(* IEC 61131-3 sources: volt/packages/volt-lsp-iec/test-corpus/lenze-mid/Device/Plc Logic/Application/Library Manager/(unresolved)/cmpopcuastack interfaces (part 4) *)

(* ---- OPCUA_BROWSENAMES.gvl ---- *)
VAR_GLOBAL
	OPCUA_BROWSENAME_3DCARTESIANCOORDINATES : STRING := '3DCartesianCoordinates';
	OPCUA_BROWSENAME_3DCARTESIANCOORDINATESTYPE : STRING := '3DCartesianCoordinatesType';
	OPCUA_BROWSENAME_3DFRAME : STRING := '3DFrame';
	OPCUA_BROWSENAME_3DFRAMETYPE : STRING := '3DFrameType';
	OPCUA_BROWSENAME_3DORIENTATION : STRING := '3DOrientation';
	OPCUA_BROWSENAME_3DORIENTATIONTYPE : STRING := '3DOrientationType';
	OPCUA_BROWSENAME_3DVECTOR : STRING := '3DVector';
	OPCUA_BROWSENAME_3DVECTORTYPE : STRING := '3DVectorType';
	OPCUA_BROWSENAME_A : STRING := 'A';
	OPCUA_BROWSENAME_ACCESSHISTORYDATACAPABILITY : STRING := 'AccessHistoryDataCapability';
	OPCUA_BROWSENAME_ACCESSHISTORYEVENTSCAPABILITY : STRING := 'AccessHistoryEventsCapability';
	OPCUA_BROWSENAME_ACCESSLEVELEXTYPE : STRING := 'AccessLevelExType';
	OPCUA_BROWSENAME_ACCESSLEVELTYPE : STRING := 'AccessLevelType';
	OPCUA_BROWSENAME_ACCESSRESTRICTIONTYPE : STRING := 'AccessRestrictionType';
	OPCUA_BROWSENAME_ACCUMULATEDLATENCY : STRING := 'AccumulatedLatency';
	OPCUA_BROWSENAME_ACKEDSTATE : STRING := 'AckedState';
	OPCUA_BROWSENAME_ACKNOWLEDGE : STRING := 'Acknowledge';
	OPCUA_BROWSENAME_ACKNOWLEDGEABLECONDITIONTYPE : STRING := 'AcknowledgeableConditionType';
	OPCUA_BROWSENAME_ACTIONTIMESTAMP : STRING := 'ActionTimeStamp';
	OPCUA_BROWSENAME_ACTIVE : STRING := 'Active';
	OPCUA_BROWSENAME_ACTIVECOUNT : STRING := 'ActiveCount';
	OPCUA_BROWSENAME_ACTIVESTATE : STRING := 'ActiveState';
	OPCUA_BROWSENAME_ACTIVITYTIMEOUT : STRING := 'ActivityTimeout';
	OPCUA_BROWSENAME_ACTUAL : STRING := 'Actual';
	OPCUA_BROWSENAME_ACTUALSESSIONTIMEOUT : STRING := 'ActualSessionTimeout';
	OPCUA_BROWSENAME_ADDAPPLICATION : STRING := 'AddApplication';
	OPCUA_BROWSENAME_ADDCERTIFICATE : STRING := 'AddCertificate';
	OPCUA_BROWSENAME_ADDCOMMENT : STRING := 'AddComment';
	OPCUA_BROWSENAME_ADDCONNECTION : STRING := 'AddConnection';
	OPCUA_BROWSENAME_ADDDATASETFOLDER : STRING := 'AddDataSetFolder';
	OPCUA_BROWSENAME_ADDDATASETREADER : STRING := 'AddDataSetReader';
	OPCUA_BROWSENAME_ADDDATASETWRITER : STRING := 'AddDataSetWriter';
	OPCUA_BROWSENAME_ADDENDPOINT : STRING := 'AddEndpoint';
	OPCUA_BROWSENAME_ADDEXTENSIONFIELD : STRING := 'AddExtensionField';
	OPCUA_BROWSENAME_ADDIDENTITY : STRING := 'AddIdentity';
	OPCUA_BROWSENAME_ADDNODESCOUNT : STRING := 'AddNodesCount';
	OPCUA_BROWSENAME_ADDNODESITEM : STRING := 'AddNodesItem';
	OPCUA_BROWSENAME_ADDPRIORITYMAPPINGENTRY : STRING := 'AddPriorityMappingEntry';
	OPCUA_BROWSENAME_ADDPUBLISHEDDATAITEMS : STRING := 'AddPublishedDataItems';
	OPCUA_BROWSENAME_ADDPUBLISHEDDATAITEMSTEMPLATE : STRING := 'AddPublishedDataItemsTemplate';
	OPCUA_BROWSENAME_ADDPUBLISHEDEVENTS : STRING := 'AddPublishedEvents';
	OPCUA_BROWSENAME_ADDPUBLISHEDEVENTSTEMPLATE : STRING := 'AddPublishedEventsTemplate';
	OPCUA_BROWSENAME_ADDPUSHTARGET : STRING := 'AddPushTarget';
	OPCUA_BROWSENAME_ADDPUSHTARGETFOLDER : STRING := 'AddPushTargetFolder';
	OPCUA_BROWSENAME_ADDREADERGROUP : STRING := 'AddReaderGroup';
	OPCUA_BROWSENAME_ADDREFERENCESCOUNT : STRING := 'AddReferencesCount';
	OPCUA_BROWSENAME_ADDREFERENCESITEM : STRING := 'AddReferencesItem';
	OPCUA_BROWSENAME_ADDROLE : STRING := 'AddRole';
	OPCUA_BROWSENAME_ADDSECURITYGROUP : STRING := 'AddSecurityGroup';
	OPCUA_BROWSENAME_ADDSECURITYGROUPFOLDER : STRING := 'AddSecurityGroupFolder';
	OPCUA_BROWSENAME_ADDSUBSCRIBEDDATASET : STRING := 'AddSubscribedDataSet';
	OPCUA_BROWSENAME_ADDTARGETVARIABLES : STRING := 'AddTargetVariables';
	OPCUA_BROWSENAME_ADDUSER : STRING := 'AddUser';
	OPCUA_BROWSENAME_ADDVARIABLES : STRING := 'AddVariables';
	OPCUA_BROWSENAME_ADDWRITERGROUP : STRING := 'AddWriterGroup';
	OPCUA_BROWSENAME_PLACEHOLDER_ADDITIONALGROUP : STRING := '<AdditionalGroup>';
	OPCUA_BROWSENAME_ADDITIONALPARAMETERSTYPE : STRING := 'AdditionalParametersType';
	OPCUA_BROWSENAME_ADDRESS : STRING := 'Address';
	OPCUA_BROWSENAME_ADDRESSSPACEFILETYPE : STRING := 'AddressSpaceFileType';
	OPCUA_BROWSENAME_ADMINSTATUS : STRING := 'AdminStatus';
	OPCUA_BROWSENAME_AFFECTEDCERTIFICATEGROUPS : STRING := 'AffectedCertificateGroups';
	OPCUA_BROWSENAME_AFFECTEDTRUSTLISTS : STRING := 'AffectedTrustLists';
	OPCUA_BROWSENAME_AGENCYID : STRING := 'AgencyId';
	OPCUA_BROWSENAME_AGGREGATECONFIGURATION : STRING := 'AggregateConfiguration';
	OPCUA_BROWSENAME_AGGREGATECONFIGURATIONTYPE : STRING := 'AggregateConfigurationType';
	OPCUA_BROWSENAME_AGGREGATEFUNCTIONTYPE : STRING := 'AggregateFunctionType';
	OPCUA_BROWSENAME_AGGREGATEFUNCTIONS : STRING := 'AggregateFunctions';
	OPCUA_BROWSENAME_AGGREGATES : STRING := 'Aggregates';
	OPCUA_BROWSENAME_PLACEHOLDER_ALARMCONDITIONINSTANCE : STRING := '<AlarmConditionInstance>';
	OPCUA_BROWSENAME_ALARMCONDITIONTYPE : STRING := 'AlarmConditionType';
	OPCUA_BROWSENAME_ALARMCOUNT : STRING := 'AlarmCount';
	OPCUA_BROWSENAME_PLACEHOLDER_ALARMGROUP : STRING := '<AlarmGroup>';
	OPCUA_BROWSENAME_ALARMGROUPMEMBER : STRING := 'AlarmGroupMember';
	OPCUA_BROWSENAME_ALARMGROUPTYPE : STRING := 'AlarmGroupType';
	OPCUA_BROWSENAME_ALARMMASK : STRING := 'AlarmMask';
	OPCUA_BROWSENAME_ALARMMETRICSTYPE : STRING := 'AlarmMetricsType';
	OPCUA_BROWSENAME_ALARMRATEVARIABLETYPE : STRING := 'AlarmRateVariableType';
	OPCUA_BROWSENAME_ALARMSTATEVARIABLETYPE : STRING := 'AlarmStateVariableType';
	OPCUA_BROWSENAME_ALARMSUPPRESSIONGROUPMEMBER : STRING := 'AlarmSuppressionGroupMember';
	OPCUA_BROWSENAME_ALARMSUPPRESSIONGROUPTYPE : STRING := 'AlarmSuppressionGroupType';
	OPCUA_BROWSENAME_PLACEHOLDER_ALIAS : STRING := '<Alias>';
	OPCUA_BROWSENAME_ALIASFOR : STRING := 'AliasFor';
	OPCUA_BROWSENAME_ALIASNAMECATEGORYTYPE : STRING := 'AliasNameCategoryType';
	OPCUA_BROWSENAME_ALIASNAMEDATATYPE : STRING := 'AliasNameDataType';
	OPCUA_BROWSENAME_ALIASNAMETYPE : STRING := 'AliasNameType';
	OPCUA_BROWSENAME_ALIASES : STRING := 'Aliases';
	OPCUA_BROWSENAME_ALLOWNULLS : STRING := 'AllowNulls';
	OPCUA_BROWSENAME_ALWAYSGENERATESEVENT : STRING := 'AlwaysGeneratesEvent';
	OPCUA_BROWSENAME_ANALOGITEMTYPE : STRING := 'AnalogItemType';
	OPCUA_BROWSENAME_ANALOGUNITRANGETYPE : STRING := 'AnalogUnitRangeType';
	OPCUA_BROWSENAME_ANALOGUNITTYPE : STRING := 'AnalogUnitType';
	OPCUA_BROWSENAME_ANGLEUNIT : STRING := 'AngleUnit';
	OPCUA_BROWSENAME_ANNOTATION : STRING := 'Annotation';
	OPCUA_BROWSENAME_ANNOTATIONCOUNT : STRING := 'AnnotationCount';
	OPCUA_BROWSENAME_ANNOTATIONS : STRING := 'Annotations';
	OPCUA_BROWSENAME_ANONYMOUS : STRING := 'Anonymous';
	OPCUA_BROWSENAME_ANONYMOUSIDENTITYTOKEN : STRING := 'AnonymousIdentityToken';
	OPCUA_BROWSENAME_APPLICATIONCERTIFICATETYPE : STRING := 'ApplicationCertificateType';
	OPCUA_BROWSENAME_APPLICATIONCONFIGURATIONTYPE : STRING := 'ApplicationConfigurationType';
	OPCUA_BROWSENAME_APPLICATIONDESCRIPTION : STRING := 'ApplicationDescription';
	OPCUA_BROWSENAME_APPLICATIONINSTANCECERTIFICATE : STRING := 'ApplicationInstanceCertificate';
	OPCUA_BROWSENAME_PLACEHOLDER_APPLICATIONNAME : STRING := '<ApplicationName>';
	OPCUA_BROWSENAME_APPLICATIONTYPE : STRING := 'ApplicationType';
	OPCUA_BROWSENAME_APPLICATIONURI : STRING := 'ApplicationUri';
	OPCUA_BROWSENAME_APPLICATIONS : STRING := 'Applications';
	OPCUA_BROWSENAME_APPLICATIONSEXCLUDE : STRING := 'ApplicationsExclude';
	OPCUA_BROWSENAME_APPLYCHANGES : STRING := 'ApplyChanges';
	OPCUA_BROWSENAME_APPLYWRITE : STRING := 'ApplyWrite';
	OPCUA_BROWSENAME_APPLYWRITETOERROR : STRING := 'ApplyWriteToError';
	OPCUA_BROWSENAME_APPLYWRITETOIDLE : STRING := 'ApplyWriteToIdle';
	OPCUA_BROWSENAME_ARGUMENT : STRING := 'Argument';
	OPCUA_BROWSENAME_ARRAYITEMTYPE : STRING := 'ArrayItemType';
	OPCUA_BROWSENAME_ASSOCIATEDWITH : STRING := 'AssociatedWith';
	OPCUA_BROWSENAME_ATTRIBUTEID : STRING := 'AttributeId';
	OPCUA_BROWSENAME_ATTRIBUTEOPERAND : STRING := 'AttributeOperand';
	OPCUA_BROWSENAME_ATTRIBUTEWRITEMASK : STRING := 'AttributeWriteMask';
	OPCUA_BROWSENAME_AUDIBLEENABLED : STRING := 'AudibleEnabled';
	OPCUA_BROWSENAME_AUDIBLESOUND : STRING := 'AudibleSound';
	OPCUA_BROWSENAME_AUDIODATATYPE : STRING := 'AudioDataType';
	OPCUA_BROWSENAME_AUDIOVARIABLETYPE : STRING := 'AudioVariableType';
	OPCUA_BROWSENAME_AUDITACTIVATESESSIONEVENTTYPE : STRING := 'AuditActivateSessionEventType';
	OPCUA_BROWSENAME_AUDITADDNODESEVENTTYPE : STRING := 'AuditAddNodesEventType';
	OPCUA_BROWSENAME_AUDITADDREFERENCESEVENTTYPE : STRING := 'AuditAddReferencesEventType';
	OPCUA_BROWSENAME_AUDITCANCELEVENTTYPE : STRING := 'AuditCancelEventType';
	OPCUA_BROWSENAME_AUDITCERTIFICATEDATAMISMATCHEVENTTYPE : STRING := 'AuditCertificateDataMismatchEventType';
	OPCUA_BROWSENAME_AUDITCERTIFICATEEVENTTYPE : STRING := 'AuditCertificateEventType';
	OPCUA_BROWSENAME_AUDITCERTIFICATEEXPIREDEVENTTYPE : STRING := 'AuditCertificateExpiredEventType';
	OPCUA_BROWSENAME_AUDITCERTIFICATEINVALIDEVENTTYPE : STRING := 'AuditCertificateInvalidEventType';
	OPCUA_BROWSENAME_AUDITCERTIFICATEMISMATCHEVENTTYPE : STRING := 'AuditCertificateMismatchEventType';
	OPCUA_BROWSENAME_AUDITCERTIFICATEREVOKEDEVENTTYPE : STRING := 'AuditCertificateRevokedEventType';
	OPCUA_BROWSENAME_AUDITCERTIFICATEUNTRUSTEDEVENTTYPE : STRING := 'AuditCertificateUntrustedEventType';
	OPCUA_BROWSENAME_AUDITCHANNELEVENTTYPE : STRING := 'AuditChannelEventType';
	OPCUA_BROWSENAME_AUDITCLIENTEVENTTYPE : STRING := 'AuditClientEventType';
	OPCUA_BROWSENAME_AUDITCLIENTUPDATEMETHODRESULTEVENTTYPE : STRING := 'AuditClientUpdateMethodResultEventType';
	OPCUA_BROWSENAME_AUDITCONDITIONACKNOWLEDGEEVENTTYPE : STRING := 'AuditConditionAcknowledgeEventType';
	OPCUA_BROWSENAME_AUDITCONDITIONCOMMENTEVENTTYPE : STRING := 'AuditConditionCommentEventType';
	OPCUA_BROWSENAME_AUDITCONDITIONCONFIRMEVENTTYPE : STRING := 'AuditConditionConfirmEventType';
	OPCUA_BROWSENAME_AUDITCONDITIONENABLEEVENTTYPE : STRING := 'AuditConditionEnableEventType';
	OPCUA_BROWSENAME_AUDITCONDITIONEVENTTYPE : STRING := 'AuditConditionEventType';
	OPCUA_BROWSENAME_AUDITCONDITIONOUTOFSERVICEEVENTTYPE : STRING := 'AuditConditionOutOfServiceEventType';
	OPCUA_BROWSENAME_AUDITCONDITIONRESETEVENTTYPE : STRING := 'AuditConditionResetEventType';
	OPCUA_BROWSENAME_AUDITCONDITIONRESPONDEVENTTYPE : STRING := 'AuditConditionRespondEventType';
	OPCUA_BROWSENAME_AUDITCONDITIONSHELVINGEVENTTYPE : STRING := 'AuditConditionShelvingEventType';
	OPCUA_BROWSENAME_AUDITCONDITIONSILENCEEVENTTYPE : STRING := 'AuditConditionSilenceEventType';
	OPCUA_BROWSENAME_AUDITCONDITIONSUPPRESSIONEVENTTYPE : STRING := 'AuditConditionSuppressionEventType';
	OPCUA_BROWSENAME_AUDITCREATESESSIONEVENTTYPE : STRING := 'AuditCreateSessionEventType';
	OPCUA_BROWSENAME_AUDITDELETENODESEVENTTYPE : STRING := 'AuditDeleteNodesEventType';
	OPCUA_BROWSENAME_AUDITDELETEREFERENCESEVENTTYPE : STRING := 'AuditDeleteReferencesEventType';
	OPCUA_BROWSENAME_AUDITEVENTTYPE : STRING := 'AuditEventType';
	OPCUA_BROWSENAME_AUDITHISTORYANNOTATIONUPDATEEVENTTYPE : STRING := 'AuditHistoryAnnotationUpdateEventType';
	OPCUA_BROWSENAME_AUDITHISTORYATTIMEDELETEEVENTTYPE : STRING := 'AuditHistoryAtTimeDeleteEventType';
	OPCUA_BROWSENAME_AUDITHISTORYDELETEEVENTTYPE : STRING := 'AuditHistoryDeleteEventType';
	OPCUA_BROWSENAME_AUDITHISTORYEVENTDELETEEVENTTYPE : STRING := 'AuditHistoryEventDeleteEventType';
	OPCUA_BROWSENAME_AUDITHISTORYEVENTUPDATEEVENTTYPE : STRING := 'AuditHistoryEventUpdateEventType';
	OPCUA_BROWSENAME_AUDITHISTORYRAWMODIFYDELETEEVENTTYPE : STRING := 'AuditHistoryRawModifyDeleteEventType';
	OPCUA_BROWSENAME_AUDITHISTORYUPDATEEVENTTYPE : STRING := 'AuditHistoryUpdateEventType';
	OPCUA_BROWSENAME_AUDITHISTORYVALUEUPDATEEVENTTYPE : STRING := 'AuditHistoryValueUpdateEventType';
	OPCUA_BROWSENAME_AUDITNODEMANAGEMENTEVENTTYPE : STRING := 'AuditNodeManagementEventType';
	OPCUA_BROWSENAME_AUDITOPENSECURECHANNELEVENTTYPE : STRING := 'AuditOpenSecureChannelEventType';
	OPCUA_BROWSENAME_AUDITPROGRAMTRANSITIONEVENTTYPE : STRING := 'AuditProgramTransitionEventType';
	OPCUA_BROWSENAME_AUDITSECURITYEVENTTYPE : STRING := 'AuditSecurityEventType';
	OPCUA_BROWSENAME_AUDITSESSIONEVENTTYPE : STRING := 'AuditSessionEventType';
	OPCUA_BROWSENAME_AUDITUPDATEEVENTTYPE : STRING := 'AuditUpdateEventType';
	OPCUA_BROWSENAME_AUDITUPDATEMETHODEVENTTYPE : STRING := 'AuditUpdateMethodEventType';
	OPCUA_BROWSENAME_AUDITUPDATESTATEEVENTTYPE : STRING := 'AuditUpdateStateEventType';
	OPCUA_BROWSENAME_AUDITURLMISMATCHEVENTTYPE : STRING := 'AuditUrlMismatchEventType';
	OPCUA_BROWSENAME_AUDITWRITEUPDATEEVENTTYPE : STRING := 'AuditWriteUpdateEventType';
	OPCUA_BROWSENAME_AUDITING : STRING := 'Auditing';
	OPCUA_BROWSENAME_AUTHENTICATEDUSER : STRING := 'AuthenticatedUser';
	OPCUA_BROWSENAME_AUTHENTICATIONMECHANISM : STRING := 'AuthenticationMechanism';
	OPCUA_BROWSENAME_AUTHENTICATIONPROFILEURI : STRING := 'AuthenticationProfileUri';
	OPCUA_BROWSENAME_AUTHORIZATIONSERVICECONFIGURATIONTYPE : STRING := 'AuthorizationServiceConfigurationType';
	OPCUA_BROWSENAME_AUTHORIZATIONSERVICES : STRING := 'AuthorizationServices';
	OPCUA_BROWSENAME_AUTHORIZATIONSERVICESCONFIGURATIONFOLDERTYPE : STRING := 'AuthorizationServicesConfigurationFolderType';
	OPCUA_BROWSENAME_AUTODELETE : STRING := 'AutoDelete';
	OPCUA_BROWSENAME_AVAILABLESTATES : STRING := 'AvailableStates';
	OPCUA_BROWSENAME_AVAILABLETRANSITIONS : STRING := 'AvailableTransitions';
	OPCUA_BROWSENAME_AVERAGE : STRING := 'Average';
	OPCUA_BROWSENAME_AVERAGEALARMRATE : STRING := 'AverageAlarmRate';
	OPCUA_BROWSENAME_AXISDEFINITION : STRING := 'AxisDefinition';
	OPCUA_BROWSENAME_AXISINFORMATION : STRING := 'AxisInformation';
	OPCUA_BROWSENAME_AXISSCALEENUMERATION : STRING := 'AxisScaleEnumeration';
	OPCUA_BROWSENAME_AXISSCALETYPE : STRING := 'AxisScaleType';
	OPCUA_BROWSENAME_B : STRING := 'B';
	OPCUA_BROWSENAME_BASEANALOGTYPE : STRING := 'BaseAnalogType';
	OPCUA_BROWSENAME_BASECONDITIONCLASSTYPE : STRING := 'BaseConditionClassType';
	OPCUA_BROWSENAME_BASEDATATYPE : STRING := 'BaseDataType';
	OPCUA_BROWSENAME_BASEDATAVARIABLETYPE : STRING := 'BaseDataVariableType';
	OPCUA_BROWSENAME_BASEEVENTTYPE : STRING := 'BaseEventType';
	OPCUA_BROWSENAME_BASEFRAME : STRING := 'BaseFrame';
	OPCUA_BROWSENAME_BASEHIGHHIGHLIMIT : STRING := 'BaseHighHighLimit';
	OPCUA_BROWSENAME_BASEHIGHLIMIT : STRING := 'BaseHighLimit';
	OPCUA_BROWSENAME_BASEINTERFACETYPE : STRING := 'BaseInterfaceType';
	OPCUA_BROWSENAME_BASELOWLIMIT : STRING := 'BaseLowLimit';
	OPCUA_BROWSENAME_BASELOWLOWLIMIT : STRING := 'BaseLowLowLimit';
	OPCUA_BROWSENAME_BASEMODELCHANGEEVENTTYPE : STRING := 'BaseModelChangeEventType';
	OPCUA_BROWSENAME_BASEOBJECTTYPE : STRING := 'BaseObjectType';
	OPCUA_BROWSENAME_BASESETPOINTNODE : STRING := 'BaseSetpointNode';
	OPCUA_BROWSENAME_BASEVARIABLETYPE : STRING := 'BaseVariableType';
	OPCUA_BROWSENAME_BITFIELDMASKDATATYPE : STRING := 'BitFieldMaskDataType';
	OPCUA_BROWSENAME_BITMASK : STRING := 'BitMask';
	OPCUA_BROWSENAME_BOOLEAN : STRING := 'Boolean';
	OPCUA_BROWSENAME_BRANCHID : STRING := 'BranchId';
	OPCUA_BROWSENAME_BROKERCONNECTIONTRANSPORTDATATYPE : STRING := 'BrokerConnectionTransportDataType';
	OPCUA_BROWSENAME_BROKERCONNECTIONTRANSPORTTYPE : STRING := 'BrokerConnectionTransportType';
	OPCUA_BROWSENAME_BROKERDATASETREADERTRANSPORTDATATYPE : STRING := 'BrokerDataSetReaderTransportDataType';
	OPCUA_BROWSENAME_BROKERDATASETREADERTRANSPORTTYPE : STRING := 'BrokerDataSetReaderTransportType';
	OPCUA_BROWSENAME_BROKERDATASETWRITERTRANSPORTDATATYPE : STRING := 'BrokerDataSetWriterTransportDataType';
	OPCUA_BROWSENAME_BROKERDATASETWRITERTRANSPORTTYPE : STRING := 'BrokerDataSetWriterTransportType';
	OPCUA_BROWSENAME_BROKERTRANSPORTQUALITYOFSERVICE : STRING := 'BrokerTransportQualityOfService';
	OPCUA_BROWSENAME_BROKERWRITERGROUPTRANSPORTDATATYPE : STRING := 'BrokerWriterGroupTransportDataType';
	OPCUA_BROWSENAME_BROKERWRITERGROUPTRANSPORTTYPE : STRING := 'BrokerWriterGroupTransportType';
	OPCUA_BROWSENAME_BROWSECOUNT : STRING := 'BrowseCount';
	OPCUA_BROWSENAME_BROWSENEXTCOUNT : STRING := 'BrowseNextCount';
	OPCUA_BROWSENAME_BUILDDATE : STRING := 'BuildDate';
	OPCUA_BROWSENAME_BUILDINFO : STRING := 'BuildInfo';
	OPCUA_BROWSENAME_BUILDINFOTYPE : STRING := 'BuildInfoType';
	OPCUA_BROWSENAME_BUILDNUMBER : STRING := 'BuildNumber';
	OPCUA_BROWSENAME_BYTE : STRING := 'Byte';
	OPCUA_BROWSENAME_BYTESTRING : STRING := 'ByteString';
	OPCUA_BROWSENAME_C : STRING := 'C';
	OPCUA_BROWSENAME_CALLCOUNT : STRING := 'CallCount';
	OPCUA_BROWSENAME_CANCELCHANGES : STRING := 'CancelChanges';
	OPCUA_BROWSENAME_CANCELRESPONSE : STRING := 'CancelResponse';
	OPCUA_BROWSENAME_CARTESIANCOORDINATES : STRING := 'CartesianCoordinates';
	OPCUA_BROWSENAME_CARTESIANCOORDINATESTYPE : STRING := 'CartesianCoordinatesType';
	OPCUA_BROWSENAME_CERTIFICATE : STRING := 'Certificate';
	OPCUA_BROWSENAME_CERTIFICATEERROREVENTID : STRING := 'CertificateErrorEventId';
	OPCUA_BROWSENAME_CERTIFICATEEXPIRATIONALARMTYPE : STRING := 'CertificateExpirationAlarmType';
	OPCUA_BROWSENAME_CERTIFICATEEXPIRED : STRING := 'CertificateExpired';
	OPCUA_BROWSENAME_CERTIFICATEGROUP : STRING := 'CertificateGroup';
	OPCUA_BROWSENAME_CERTIFICATEGROUPFOLDERTYPE : STRING := 'CertificateGroupFolderType';
	OPCUA_BROWSENAME_CERTIFICATEGROUPTYPE : STRING := 'CertificateGroupType';
	OPCUA_BROWSENAME_CERTIFICATEGROUPS : STRING := 'CertificateGroups';
	OPCUA_BROWSENAME_CERTIFICATETYPE : STRING := 'CertificateType';
	OPCUA_BROWSENAME_CERTIFICATETYPES : STRING := 'CertificateTypes';
	OPCUA_BROWSENAME_CERTIFICATEUPDATEREQUESTEDAUDITEVENTTYPE : STRING := 'CertificateUpdateRequestedAuditEventType';
	OPCUA_BROWSENAME_CERTIFICATEUPDATEDAUDITEVENTTYPE : STRING := 'CertificateUpdatedAuditEventType';
	OPCUA_BROWSENAME_CHANGEPASSWORD : STRING := 'ChangePassword';
	OPCUA_BROWSENAME_CHANGES : STRING := 'Changes';
	OPCUA_BROWSENAME_CHOICESTATETYPE : STRING := 'ChoiceStateType';
	OPCUA_BROWSENAME_CLASSIFICATION : STRING := 'Classification';
	OPCUA_BROWSENAME_CLIENTAUDITENTRYID : STRING := 'ClientAuditEntryId';
	OPCUA_BROWSENAME_CLIENTCERTIFICATE : STRING := 'ClientCertificate';
	OPCUA_BROWSENAME_CLIENTCERTIFICATETHUMBPRINT : STRING := 'ClientCertificateThumbprint';
	OPCUA_BROWSENAME_CLIENTCONNECTIONTIME : STRING := 'ClientConnectionTime';
	OPCUA_BROWSENAME_CLIENTDESCRIPTION : STRING := 'ClientDescription';
	OPCUA_BROWSENAME_CLIENTLASTCONTACTTIME : STRING := 'ClientLastContactTime';
	OPCUA_BROWSENAME_PLACEHOLDER_CLIENTNAME : STRING := '<ClientName>';
	OPCUA_BROWSENAME_CLIENTPROCESSINGTIMEOUT : STRING := 'ClientProcessingTimeout';
	OPCUA_BROWSENAME_CLIENTSOFTWARECERTIFICATES : STRING := 'ClientSoftwareCertificates';
	OPCUA_BROWSENAME_CLIENTUSERID : STRING := 'ClientUserId';
	OPCUA_BROWSENAME_CLIENTUSERIDHISTORY : STRING := 'ClientUserIdHistory';
	OPCUA_BROWSENAME_CLIENTUSERIDOFSESSION : STRING := 'ClientUserIdOfSession';
	OPCUA_BROWSENAME_CLOSE : STRING := 'Close';
	OPCUA_BROWSENAME_CLOSEANDCOMMIT : STRING := 'CloseAndCommit';
	OPCUA_BROWSENAME_CLOSEANDUPDATE : STRING := 'CloseAndUpdate';
	OPCUA_BROWSENAME_COMMENT : STRING := 'Comment';
	OPCUA_BROWSENAME_COMMUNICATION : STRING := 'Communication';
	OPCUA_BROWSENAME_COMPLEXNUMBERTYPE : STRING := 'ComplexNumberType';
	OPCUA_BROWSENAME_CONDITIONCLASSID : STRING := 'ConditionClassId';
	OPCUA_BROWSENAME_CONDITIONCLASSNAME : STRING := 'ConditionClassName';
	OPCUA_BROWSENAME_CONDITIONEVENTID : STRING := 'ConditionEventId';
	OPCUA_BROWSENAME_CONDITIONNAME : STRING := 'ConditionName';
	OPCUA_BROWSENAME_CONDITIONREFRESH : STRING := 'ConditionRefresh';
	OPCUA_BROWSENAME_CONDITIONREFRESH2 : STRING := 'ConditionRefresh2';
	OPCUA_BROWSENAME_CONDITIONSUBCLASSID : STRING := 'ConditionSubClassId';
	OPCUA_BROWSENAME_CONDITIONSUBCLASSNAME : STRING := 'ConditionSubClassName';
	OPCUA_BROWSENAME_CONDITIONTYPE : STRING := 'ConditionType';
	OPCUA_BROWSENAME_CONDITIONVARIABLETYPE : STRING := 'ConditionVariableType';
	OPCUA_BROWSENAME_CONFIGURATIONPROPERTIES : STRING := 'ConfigurationProperties';
	OPCUA_BROWSENAME_CONFIGURATIONVERSION : STRING := 'ConfigurationVersion';
	OPCUA_BROWSENAME_CONFIGURATIONVERSIONDATATYPE : STRING := 'ConfigurationVersionDataType';
	OPCUA_BROWSENAME_CONFIGUREADMIN : STRING := 'ConfigureAdmin';
	OPCUA_BROWSENAME_CONFIGUREDDATASETREADERS : STRING := 'ConfiguredDataSetReaders';
	OPCUA_BROWSENAME_CONFIGUREDDATASETWRITERS : STRING := 'ConfiguredDataSetWriters';
	OPCUA_BROWSENAME_CONFIGUREDSIZE : STRING := 'ConfiguredSize';
	OPCUA_BROWSENAME_CONFIRM : STRING := 'Confirm';
	OPCUA_BROWSENAME_CONFIRMEDSTATE : STRING := 'ConfirmedState';
	OPCUA_BROWSENAME_CONFORMANCEUNITS : STRING := 'ConformanceUnits';
	OPCUA_BROWSENAME_CONNECTSECURITYGROUPS : STRING := 'ConnectSecurityGroups';
	OPCUA_BROWSENAME_CONNECTIONID : STRING := 'ConnectionId';
	OPCUA_BROWSENAME_PLACEHOLDER_CONNECTIONNAME : STRING := '<ConnectionName>';
	OPCUA_BROWSENAME_CONNECTIONPROPERTIES : STRING := 'ConnectionProperties';
	OPCUA_BROWSENAME_CONNECTIONTRANSPORTDATATYPE : STRING := 'ConnectionTransportDataType';
	OPCUA_BROWSENAME_CONNECTIONTRANSPORTTYPE : STRING := 'ConnectionTransportType';
	OPCUA_BROWSENAME_CONSTANT : STRING := 'Constant';
	OPCUA_BROWSENAME_CONTENTFILTER : STRING := 'ContentFilter';
	OPCUA_BROWSENAME_CONTENTFILTERELEMENT : STRING := 'ContentFilterElement';
	OPCUA_BROWSENAME_CONTEXT : STRING := 'Context';
	OPCUA_BROWSENAME_CONTINUATIONPOINT : STRING := 'ContinuationPoint';
	OPCUA_BROWSENAME_CONTROLS : STRING := 'Controls';
	OPCUA_BROWSENAME_COUNT : STRING := 'Count';
	OPCUA_BROWSENAME_COUNTER : STRING := 'Counter';
	OPCUA_BROWSENAME_COUNTERS : STRING := 'Counters';
	OPCUA_BROWSENAME_CREATABLE : STRING := 'Creatable';
	OPCUA_BROWSENAME_CREATECLIENTNAME : STRING := 'CreateClientName';
	OPCUA_BROWSENAME_CREATECREDENTIAL : STRING := 'CreateCredential';
	OPCUA_BROWSENAME_CREATEDATASETMIRROR : STRING := 'CreateDataSetMirror';
	OPCUA_BROWSENAME_CREATEDIRECTORY : STRING := 'CreateDirectory';
	OPCUA_BROWSENAME_CREATEFILE : STRING := 'CreateFile';
	OPCUA_BROWSENAME_CREATEMONITOREDITEMSCOUNT : STRING := 'CreateMonitoredItemsCount';
	OPCUA_BROWSENAME_CREATESESSIONID : STRING := 'CreateSessionId';
	OPCUA_BROWSENAME_CREATESIGNINGREQUEST : STRING := 'CreateSigningRequest';
	OPCUA_BROWSENAME_CREATESUBSCRIPTIONCOUNT : STRING := 'CreateSubscriptionCount';
	OPCUA_BROWSENAME_CREATETARGETVARIABLES : STRING := 'CreateTargetVariables';
	OPCUA_BROWSENAME_CUBEITEMTYPE : STRING := 'CubeItemType';
	OPCUA_BROWSENAME_CUMULATEDSESSIONCOUNT : STRING := 'CumulatedSessionCount';
	OPCUA_BROWSENAME_CUMULATEDSUBSCRIPTIONCOUNT : STRING := 'CumulatedSubscriptionCount';
	OPCUA_BROWSENAME_CURRENCYUNIT : STRING := 'CurrencyUnit';
	OPCUA_BROWSENAME_CURRENCYUNITTYPE : STRING := 'CurrencyUnitType';
	OPCUA_BROWSENAME_CURRENTALARMRATE : STRING := 'CurrentAlarmRate';
	OPCUA_BROWSENAME_CURRENTKEEPALIVECOUNT : STRING := 'CurrentKeepAliveCount';
	OPCUA_BROWSENAME_CURRENTLIFETIMECOUNT : STRING := 'CurrentLifetimeCount';
	OPCUA_BROWSENAME_CURRENTMONITOREDITEMSCOUNT : STRING := 'CurrentMonitoredItemsCount';
	OPCUA_BROWSENAME_CURRENTPUBLISHREQUESTSINQUEUE : STRING := 'CurrentPublishRequestsInQueue';
	OPCUA_BROWSENAME_CURRENTSERVERID : STRING := 'CurrentServerId';
	OPCUA_BROWSENAME_CURRENTSESSIONCOUNT : STRING := 'CurrentSessionCount';
	OPCUA_BROWSENAME_CURRENTSTATE : STRING := 'CurrentState';
	OPCUA_BROWSENAME_CURRENTSUBSCRIPTIONCOUNT : STRING := 'CurrentSubscriptionCount';
	OPCUA_BROWSENAME_CURRENTSUBSCRIPTIONSCOUNT : STRING := 'CurrentSubscriptionsCount';
	OPCUA_BROWSENAME_CURRENTTIME : STRING := 'CurrentTime';
	OPCUA_BROWSENAME_CUSTOMCONFIGURATION : STRING := 'CustomConfiguration';
	OPCUA_BROWSENAME_CYCLICDATASET : STRING := 'CyclicDataSet';
	OPCUA_BROWSENAME_DATACHANGENOTIFICATIONSCOUNT : STRING := 'DataChangeNotificationsCount';
	OPCUA_BROWSENAME_DATAITEMTYPE : STRING := 'DataItemType';
	OPCUA_BROWSENAME_DATASETCLASSID : STRING := 'DataSetClassId';
	OPCUA_BROWSENAME_DATASETCLASSES : STRING := 'DataSetClasses';
	OPCUA_BROWSENAME_DATASETFIELDCONTENTMASK : STRING := 'DataSetFieldContentMask';
	OPCUA_BROWSENAME_DATASETFIELDFLAGS : STRING := 'DataSetFieldFlags';
	OPCUA_BROWSENAME_PLACEHOLDER_DATASETFOLDERNAME : STRING := '<DataSetFolderName>';
	OPCUA_BROWSENAME_DATASETFOLDERTYPE : STRING := 'DataSetFolderType';
	OPCUA_BROWSENAME_DATASETMESSAGECONTENTMASK : STRING := 'DataSetMessageContentMask';
	OPCUA_BROWSENAME_DATASETMETADATA : STRING := 'DataSetMetaData';
	OPCUA_BROWSENAME_DATASETMETADATATYPE : STRING := 'DataSetMetaDataType';
	OPCUA_BROWSENAME_PLACEHOLDER_DATASETNAME : STRING := '<DataSetName>';
	OPCUA_BROWSENAME_DATASETOFFSET : STRING := 'DataSetOffset';
	OPCUA_BROWSENAME_DATASETORDERING : STRING := 'DataSetOrdering';
	OPCUA_BROWSENAME_DATASETORDERINGTYPE : STRING := 'DataSetOrderingType';
	OPCUA_BROWSENAME_DATASETREADERDATATYPE : STRING := 'DataSetReaderDataType';
	OPCUA_BROWSENAME_DATASETREADERMESSAGEDATATYPE : STRING := 'DataSetReaderMessageDataType';
	OPCUA_BROWSENAME_DATASETREADERMESSAGETYPE : STRING := 'DataSetReaderMessageType';
	OPCUA_BROWSENAME_PLACEHOLDER_DATASETREADERNAME : STRING := '<DataSetReaderName>';
	OPCUA_BROWSENAME_DATASETREADERPROPERTIES : STRING := 'DataSetReaderProperties';
	OPCUA_BROWSENAME_DATASETREADERTRANSPORTDATATYPE : STRING := 'DataSetReaderTransportDataType';
	OPCUA_BROWSENAME_DATASETREADERTRANSPORTTYPE : STRING := 'DataSetReaderTransportType';
	OPCUA_BROWSENAME_DATASETREADERTYPE : STRING := 'DataSetReaderType';
	OPCUA_BROWSENAME_DATASETTOWRITER : STRING := 'DataSetToWriter';
	OPCUA_BROWSENAME_DATASETWRITERDATATYPE : STRING := 'DataSetWriterDataType';
	OPCUA_BROWSENAME_DATASETWRITERID : STRING := 'DataSetWriterId';
	OPCUA_BROWSENAME_DATASETWRITERMESSAGEDATATYPE : STRING := 'DataSetWriterMessageDataType';
	OPCUA_BROWSENAME_DATASETWRITERMESSAGETYPE : STRING := 'DataSetWriterMessageType';
	OPCUA_BROWSENAME_PLACEHOLDER_DATASETWRITERNAME : STRING := '<DataSetWriterName>';
	OPCUA_BROWSENAME_DATASETWRITERPROPERTIES : STRING := 'DataSetWriterProperties';
	OPCUA_BROWSENAME_DATASETWRITERTRANSPORTDATATYPE : STRING := 'DataSetWriterTransportDataType';
	OPCUA_BROWSENAME_DATASETWRITERTRANSPORTTYPE : STRING := 'DataSetWriterTransportType';
	OPCUA_BROWSENAME_DATASETWRITERTYPE : STRING := 'DataSetWriterType';
	OPCUA_BROWSENAME_DATATYPEDEFINITION : STRING := 'DataTypeDefinition';
	OPCUA_BROWSENAME_DATATYPEDESCRIPTION : STRING := 'DataTypeDescription';
	OPCUA_BROWSENAME_DATATYPEDESCRIPTIONTYPE : STRING := 'DataTypeDescriptionType';
	OPCUA_BROWSENAME_DATATYPEDICTIONARYTYPE : STRING := 'DataTypeDictionaryType';
	OPCUA_BROWSENAME_DATATYPEENCODINGTYPE : STRING := 'DataTypeEncodingType';
	OPCUA_BROWSENAME_DATATYPESCHEMAHEADER : STRING := 'DataTypeSchemaHeader';
	OPCUA_BROWSENAME_DATATYPESYSTEMTYPE : STRING := 'DataTypeSystemType';
	OPCUA_BROWSENAME_DATATYPEVERSION : STRING := 'DataTypeVersion';
	OPCUA_BROWSENAME_DATATYPES : STRING := 'DataTypes';
	OPCUA_BROWSENAME_DATAVALUE : STRING := 'DataValue';
	OPCUA_BROWSENAME_DATAGRAMCONNECTIONTRANSPORT2DATATYPE : STRING := 'DatagramConnectionTransport2DataType';
	OPCUA_BROWSENAME_DATAGRAMCONNECTIONTRANSPORTDATATYPE : STRING := 'DatagramConnectionTransportDataType';
	OPCUA_BROWSENAME_DATAGRAMCONNECTIONTRANSPORTTYPE : STRING := 'DatagramConnectionTransportType';
	OPCUA_BROWSENAME_DATAGRAMDATASETREADERTRANSPORTDATATYPE : STRING := 'DatagramDataSetReaderTransportDataType';
	OPCUA_BROWSENAME_DATAGRAMDATASETREADERTRANSPORTTYPE : STRING := 'DatagramDataSetReaderTransportType';
	OPCUA_BROWSENAME_DATAGRAMQOS : STRING := 'DatagramQos';
	OPCUA_BROWSENAME_DATAGRAMWRITERGROUPTRANSPORT2DATATYPE : STRING := 'DatagramWriterGroupTransport2DataType';
	OPCUA_BROWSENAME_DATAGRAMWRITERGROUPTRANSPORTDATATYPE : STRING := 'DatagramWriterGroupTransportDataType';
	OPCUA_BROWSENAME_DATAGRAMWRITERGROUPTRANSPORTTYPE : STRING := 'DatagramWriterGroupTransportType';
	OPCUA_BROWSENAME_DATESTRING : STRING := 'DateString';
	OPCUA_BROWSENAME_DATETIME : STRING := 'DateTime';
	OPCUA_BROWSENAME_DECIMAL : STRING := 'Decimal';
	OPCUA_BROWSENAME_DECIMALSTRING : STRING := 'DecimalString';
	OPCUA_BROWSENAME_DECRYPTIONERRORS : STRING := 'DecryptionErrors';
	OPCUA_BROWSENAME_DEFAULTBINARY : STRING := 'Default Binary';
	OPCUA_BROWSENAME_DEFAULTJSON : STRING := 'Default JSON';
	OPCUA_BROWSENAME_DEFAULTXML : STRING := 'Default XML';
	OPCUA_BROWSENAME_DEFAULTACCESSRESTRICTIONS : STRING := 'DefaultAccessRestrictions';
	OPCUA_BROWSENAME_DEFAULTAPPLICATIONGROUP : STRING := 'DefaultApplicationGroup';
	OPCUA_BROWSENAME_DEFAULTDATAGRAMPUBLISHERID : STRING := 'DefaultDatagramPublisherId';
	OPCUA_BROWSENAME_DEFAULTHTTPSGROUP : STRING := 'DefaultHttpsGroup';
	OPCUA_BROWSENAME_DEFAULTINSTANCEBROWSENAME : STRING := 'DefaultInstanceBrowseName';
	OPCUA_BROWSENAME_DEFAULTRESPONSE : STRING := 'DefaultResponse';
	OPCUA_BROWSENAME_DEFAULTROLEPERMISSIONS : STRING := 'DefaultRolePermissions';
	OPCUA_BROWSENAME_DEFAULTSECURITYKEYSERVICES : STRING := 'DefaultSecurityKeyServices';
	OPCUA_BROWSENAME_DEFAULTUSERROLEPERMISSIONS : STRING := 'DefaultUserRolePermissions';
	OPCUA_BROWSENAME_DEFAULTUSERTOKENGROUP : STRING := 'DefaultUserTokenGroup';
	OPCUA_BROWSENAME_DEFAULTVALIDATIONOPTIONS : STRING := 'DefaultValidationOptions';
	OPCUA_BROWSENAME_DEFINITION : STRING := 'Definition';
	OPCUA_BROWSENAME_DELETABLE : STRING := 'Deletable';
	OPCUA_BROWSENAME_DELETE : STRING := 'Delete';
	OPCUA_BROWSENAME_DELETEATTIMECAPABILITY : STRING := 'DeleteAtTimeCapability';
	OPCUA_BROWSENAME_DELETECREDENTIAL : STRING := 'DeleteCredential';
	OPCUA_BROWSENAME_DELETEEVENTCAPABILITY : STRING := 'DeleteEventCapability';
	OPCUA_BROWSENAME_DELETEMONITOREDITEMSCOUNT : STRING := 'DeleteMonitoredItemsCount';
	OPCUA_BROWSENAME_DELETENODESCOUNT : STRING := 'DeleteNodesCount';
	OPCUA_BROWSENAME_DELETENODESITEM : STRING := 'DeleteNodesItem';
	OPCUA_BROWSENAME_DELETEPRIORITYMAPPINGENTRY : STRING := 'DeletePriorityMappingEntry';
	OPCUA_BROWSENAME_DELETERAWCAPABILITY : STRING := 'DeleteRawCapability';
	OPCUA_BROWSENAME_DELETEREFERENCESCOUNT : STRING := 'DeleteReferencesCount';
	OPCUA_BROWSENAME_DELETEREFERENCESITEM : STRING := 'DeleteReferencesItem';
	OPCUA_BROWSENAME_DELETESUBSCRIPTIONSCOUNT : STRING := 'DeleteSubscriptionsCount';
	OPCUA_BROWSENAME_DELTA : STRING := 'Delta';
	OPCUA_BROWSENAME_DELTABOUNDS : STRING := 'DeltaBounds';
	OPCUA_BROWSENAME_DENOMINATOR : STRING := 'Denominator';
	OPCUA_BROWSENAME_DEPRECATED : STRING := 'Deprecated';
	OPCUA_BROWSENAME_DESTINATIONADDRESS : STRING := 'DestinationAddress';
	OPCUA_BROWSENAME_DEVICEFAILUREEVENTTYPE : STRING := 'DeviceFailureEventType';
	OPCUA_BROWSENAME_DIAGNOSTICINFO : STRING := 'DiagnosticInfo';
	OPCUA_BROWSENAME_DIAGNOSTICS : STRING := 'Diagnostics';
	OPCUA_BROWSENAME_DIAGNOSTICSLEVEL : STRING := 'DiagnosticsLevel';
	OPCUA_BROWSENAME_DIALOGCONDITIONTYPE : STRING := 'DialogConditionType';
	OPCUA_BROWSENAME_DIALOGSTATE : STRING := 'DialogState';
	OPCUA_BROWSENAME_DICTIONARIES : STRING := 'Dictionaries';
	OPCUA_BROWSENAME_PLACEHOLDER_DICTIONARYENTRYNAME : STRING := '<DictionaryEntryName>';
	OPCUA_BROWSENAME_DICTIONARYENTRYTYPE : STRING := 'DictionaryEntryType';
	OPCUA_BROWSENAME_PLACEHOLDER_DICTIONARYFOLDERNAME : STRING := '<DictionaryFolderName>';
	OPCUA_BROWSENAME_DICTIONARYFOLDERTYPE : STRING := 'DictionaryFolderType';
	OPCUA_BROWSENAME_DICTIONARYFRAGMENT : STRING := 'DictionaryFragment';
	OPCUA_BROWSENAME_PLACEHOLDER_DIGITALVARIABLE : STRING := '<DigitalVariable>';
	OPCUA_BROWSENAME_DISABLE : STRING := 'Disable';
	OPCUA_BROWSENAME_DISABLECOUNT : STRING := 'DisableCount';
	OPCUA_BROWSENAME_DISABLEDMONITOREDITEMCOUNT : STRING := 'DisabledMonitoredItemCount';
	OPCUA_BROWSENAME_DISABLEDMONITOREDITEMSSAMPLINGCOUNT : STRING := 'DisabledMonitoredItemsSamplingCount';
	OPCUA_BROWSENAME_DISCARDEDMESSAGECOUNT : STRING := 'DiscardedMessageCount';
	OPCUA_BROWSENAME_DISCONNECTSECURITYGROUPS : STRING := 'DisconnectSecurityGroups';
	OPCUA_BROWSENAME_DISCOVERYADDRESS : STRING := 'DiscoveryAddress';
	OPCUA_BROWSENAME_DISCOVERYANNOUNCERATE : STRING := 'DiscoveryAnnounceRate';
	OPCUA_BROWSENAME_DISCOVERYCONFIGURATION : STRING := 'DiscoveryConfiguration';
	OPCUA_BROWSENAME_DISCOVERYMAXMESSAGESIZE : STRING := 'DiscoveryMaxMessageSize';
	OPCUA_BROWSENAME_DISCREPANCYALARMTYPE : STRING := 'DiscrepancyAlarmType';
	OPCUA_BROWSENAME_DISCRETEALARMTYPE : STRING := 'DiscreteAlarmType';
	OPCUA_BROWSENAME_DISCRETEITEMTYPE : STRING := 'DiscreteItemType';
	OPCUA_BROWSENAME_DOUBLE : STRING := 'Double';
	OPCUA_BROWSENAME_DOUBLECOMPLEXNUMBERTYPE : STRING := 'DoubleComplexNumberType';
	OPCUA_BROWSENAME_DUPLEX : STRING := 'Duplex';
	OPCUA_BROWSENAME_DURATION : STRING := 'Duration';
	OPCUA_BROWSENAME_DURATIONBAD : STRING := 'DurationBad';
	OPCUA_BROWSENAME_DURATIONGOOD : STRING := 'DurationGood';
	OPCUA_BROWSENAME_DURATIONINSTATENONZERO : STRING := 'DurationInStateNonZero';
	OPCUA_BROWSENAME_DURATIONINSTATEZERO : STRING := 'DurationInStateZero';
	OPCUA_BROWSENAME_DURATIONSTRING : STRING := 'DurationString';
	OPCUA_BROWSENAME_EUINFORMATION : STRING := 'EUInformation';
	OPCUA_BROWSENAME_EURANGE : STRING := 'EURange';
	OPCUA_BROWSENAME_ECCAPPLICATIONCERTIFICATETYPE : STRING := 'EccApplicationCertificateType';
	OPCUA_BROWSENAME_ECCBRAINPOOLP256R1APPLICATIONCERTIFICATETYPE : STRING := 'EccBrainpoolP256r1ApplicationCertificateType';
	OPCUA_BROWSENAME_ECCBRAINPOOLP384R1APPLICATIONCERTIFICATETYPE : STRING := 'EccBrainpoolP384r1ApplicationCertificateType';
	OPCUA_BROWSENAME_ECCCURVE25519APPLICATIONCERTIFICATETYPE : STRING := 'EccCurve25519ApplicationCertificateType';
	OPCUA_BROWSENAME_ECCCURVE448APPLICATIONCERTIFICATETYPE : STRING := 'EccCurve448ApplicationCertificateType';
	OPCUA_BROWSENAME_ECCNISTP256APPLICATIONCERTIFICATETYPE : STRING := 'EccNistP256ApplicationCertificateType';
	OPCUA_BROWSENAME_ECCNISTP384APPLICATIONCERTIFICATETYPE : STRING := 'EccNistP384ApplicationCertificateType';
	OPCUA_BROWSENAME_EFFECTIVEDISPLAYNAME : STRING := 'EffectiveDisplayName';
	OPCUA_BROWSENAME_EFFECTIVETRANSITIONTIME : STRING := 'EffectiveTransitionTime';
	OPCUA_BROWSENAME_ELEMENTOPERAND : STRING := 'ElementOperand';
	OPCUA_BROWSENAME_ELSEGUARDVARIABLETYPE : STRING := 'ElseGuardVariableType';
	OPCUA_BROWSENAME_ENABLE : STRING := 'Enable';
	OPCUA_BROWSENAME_ENABLECOUNT : STRING := 'EnableCount';
	OPCUA_BROWSENAME_ENABLED : STRING := 'Enabled';
	OPCUA_BROWSENAME_ENABLEDFLAG : STRING := 'EnabledFlag';
	OPCUA_BROWSENAME_ENABLEDSTATE : STRING := 'EnabledState';
	OPCUA_BROWSENAME_ENCODEDTICKET : STRING := 'EncodedTicket';
	OPCUA_BROWSENAME_ENCODING : STRING := 'Encoding';
	OPCUA_BROWSENAME_ENCRYPTIONERRORS : STRING := 'EncryptionErrors';
	OPCUA_BROWSENAME_END : STRING := 'End';
	OPCUA_BROWSENAME_ENDBOUND : STRING := 'EndBound';
	OPCUA_BROWSENAME_ENDTIME : STRING := 'EndTime';
	OPCUA_BROWSENAME_ENDPOINTCONFIGURATION : STRING := 'EndpointConfiguration';
	OPCUA_BROWSENAME_ENDPOINTDESCRIPTION : STRING := 'EndpointDescription';
	OPCUA_BROWSENAME_ENDPOINTTYPE : STRING := 'EndpointType';
	OPCUA_BROWSENAME_ENDPOINTURL : STRING := 'EndpointUrl';
	OPCUA_BROWSENAME_ENDPOINTURLLISTDATATYPE : STRING := 'EndpointUrlListDataType';
	OPCUA_BROWSENAME_ENDPOINTURLS : STRING := 'EndpointUrls';
	OPCUA_BROWSENAME_ENDPOINTS : STRING := 'Endpoints';
	OPCUA_BROWSENAME_ENDPOINTSEXCLUDE : STRING := 'EndpointsExclude';
	OPCUA_BROWSENAME_ENGINEER : STRING := 'Engineer';
	OPCUA_BROWSENAME_ENGINEERINGUNITS : STRING := 'EngineeringUnits';
	OPCUA_BROWSENAME_ENUMDEFINITION : STRING := 'EnumDefinition';
	OPCUA_BROWSENAME_ENUMDESCRIPTION : STRING := 'EnumDescription';
	OPCUA_BROWSENAME_ENUMDICTIONARYENTRIES : STRING := 'EnumDictionaryEntries';
	OPCUA_BROWSENAME_ENUMFIELD : STRING := 'EnumField';
	OPCUA_BROWSENAME_ENUMSTRINGS : STRING := 'EnumStrings';
	OPCUA_BROWSENAME_ENUMVALUETYPE : STRING := 'EnumValueType';
	OPCUA_BROWSENAME_ENUMVALUES : STRING := 'EnumValues';
	OPCUA_BROWSENAME_ENUMERATION : STRING := 'Enumeration';
	OPCUA_BROWSENAME_EPHEMERALKEYTYPE : STRING := 'EphemeralKeyType';
	OPCUA_BROWSENAME_ERROR : STRING := 'Error';
	OPCUA_BROWSENAME_ERRORTOIDLE : STRING := 'ErrorToIdle';
	OPCUA_BROWSENAME_ERRORS : STRING := 'Errors';
	OPCUA_BROWSENAME_ESTIMATEDRETURNTIME : STRING := 'EstimatedReturnTime';
	OPCUA_BROWSENAME_EVENTFILTER : STRING := 'EventFilter';
	OPCUA_BROWSENAME_EVENTID : STRING := 'EventId';
	OPCUA_BROWSENAME_EVENTIDS : STRING := 'EventIds';
	OPCUA_BROWSENAME_EVENTNOTIFICATIONSCOUNT : STRING := 'EventNotificationsCount';
	OPCUA_BROWSENAME_EVENTNOTIFIER : STRING := 'EventNotifier';
	OPCUA_BROWSENAME_EVENTNOTIFIERTYPE : STRING := 'EventNotifierType';
	OPCUA_BROWSENAME_EVENTQUEUEOVERFLOWCOUNT : STRING := 'EventQueueOverflowCount';
	OPCUA_BROWSENAME_EVENTQUEUEOVERFLOWEVENTTYPE : STRING := 'EventQueueOverflowEventType';
	OPCUA_BROWSENAME_EVENTTYPE : STRING := 'EventType';
	OPCUA_BROWSENAME_EVENTTYPES : STRING := 'EventTypes';
	OPCUA_BROWSENAME_EXCEPTIONDEVIATION : STRING := 'ExceptionDeviation';
	OPCUA_BROWSENAME_EXCEPTIONDEVIATIONFORMAT : STRING := 'ExceptionDeviationFormat';
	OPCUA_BROWSENAME_EXCLUSIVEDEVIATIONALARMTYPE : STRING := 'ExclusiveDeviationAlarmType';
	OPCUA_BROWSENAME_EXCLUSIVELEVELALARMTYPE : STRING := 'ExclusiveLevelAlarmType';
	OPCUA_BROWSENAME_EXCLUSIVELIMITALARMTYPE : STRING := 'ExclusiveLimitAlarmType';
	OPCUA_BROWSENAME_EXCLUSIVELIMITSTATEMACHINETYPE : STRING := 'ExclusiveLimitStateMachineType';
	OPCUA_BROWSENAME_EXCLUSIVERATEOFCHANGEALARMTYPE : STRING := 'ExclusiveRateOfChangeAlarmType';
	OPCUA_BROWSENAME_EXPANDEDNODEID : STRING := 'ExpandedNodeId';
	OPCUA_BROWSENAME_EXPECTEDTIME : STRING := 'ExpectedTime';
	OPCUA_BROWSENAME_EXPIRATIONDATE : STRING := 'ExpirationDate';
	OPCUA_BROWSENAME_EXPIRATIONLIMIT : STRING := 'ExpirationLimit';
	OPCUA_BROWSENAME_EXPORTNAMESPACE : STRING := 'ExportNamespace';
	OPCUA_BROWSENAME_EXPOSESITSARRAY : STRING := 'ExposesItsArray';
	OPCUA_BROWSENAME_EXPRESSION : STRING := 'Expression';
	OPCUA_BROWSENAME_EXPRESSIONGUARDVARIABLETYPE : STRING := 'ExpressionGuardVariableType';
	OPCUA_BROWSENAME_PLACEHOLDER_EXTENSIONFIELDNAME : STRING := '<ExtensionFieldName>';
	OPCUA_BROWSENAME_EXTENSIONFIELDS : STRING := 'ExtensionFields';
	OPCUA_BROWSENAME_EXTENSIONFIELDSTYPE : STRING := 'ExtensionFieldsType';
	OPCUA_BROWSENAME_FAILEDDATASETMESSAGES : STRING := 'FailedDataSetMessages';
	OPCUA_BROWSENAME_FAILEDTRANSMISSIONS : STRING := 'FailedTransmissions';
	OPCUA_BROWSENAME_FAILURECODE : STRING := 'FailureCode';
	OPCUA_BROWSENAME_FAILURESYSTEMIDENTIFIER : STRING := 'FailureSystemIdentifier';
	OPCUA_BROWSENAME_FALSESTATE : STRING := 'FalseState';
	OPCUA_BROWSENAME_FIELDMETADATA : STRING := 'FieldMetaData';
	OPCUA_BROWSENAME_FIELDTARGETDATATYPE : STRING := 'FieldTargetDataType';
	OPCUA_BROWSENAME_PLACEHOLDER_FILEDIRECTORYNAME : STRING := '<FileDirectoryName>';
	OPCUA_BROWSENAME_FILEDIRECTORYTYPE : STRING := 'FileDirectoryType';
	OPCUA_BROWSENAME_PLACEHOLDER_FILENAME : STRING := '<FileName>';
	OPCUA_BROWSENAME_FILESYSTEM : STRING := 'FileSystem';
	OPCUA_BROWSENAME_FILETRANSFERSTATEMACHINETYPE : STRING := 'FileTransferStateMachineType';
	OPCUA_BROWSENAME_FILETYPE : STRING := 'FileType';
	OPCUA_BROWSENAME_FILTER : STRING := 'Filter';
	OPCUA_BROWSENAME_FILTEROPERAND : STRING := 'FilterOperand';
	OPCUA_BROWSENAME_FILTEROPERATOR : STRING := 'FilterOperator';
	OPCUA_BROWSENAME_FINALRESULTDATA : STRING := 'FinalResultData';
	OPCUA_BROWSENAME_FINDALIAS : STRING := 'FindAlias';
	OPCUA_BROWSENAME_FINITESTATEMACHINETYPE : STRING := 'FiniteStateMachineType';
	OPCUA_BROWSENAME_FINITESTATEVARIABLETYPE : STRING := 'FiniteStateVariableType';
	OPCUA_BROWSENAME_FINITETRANSITIONVARIABLETYPE : STRING := 'FiniteTransitionVariableType';
	OPCUA_BROWSENAME_FIRSTINGROUP : STRING := 'FirstInGroup';
	OPCUA_BROWSENAME_FIRSTINGROUPFLAG : STRING := 'FirstInGroupFlag';
	OPCUA_BROWSENAME_FIXEDBASE : STRING := 'FixedBase';
	OPCUA_BROWSENAME_FLOAT : STRING := 'Float';
	OPCUA_BROWSENAME_FOLDERTYPE : STRING := 'FolderType';
	OPCUA_BROWSENAME_FORCEKEYROTATION : STRING := 'ForceKeyRotation';
	OPCUA_BROWSENAME_FRAME : STRING := 'Frame';
	OPCUA_BROWSENAME_FRAMETYPE : STRING := 'FrameType';
	OPCUA_BROWSENAME_FROMSTATE : STRING := 'FromState';
	OPCUA_BROWSENAME_GENERALMODELCHANGEEVENTTYPE : STRING := 'GeneralModelChangeEventType';
	OPCUA_BROWSENAME_GENERATEFILEFORREAD : STRING := 'GenerateFileForRead';
	OPCUA_BROWSENAME_GENERATEFILEFORWRITE : STRING := 'GenerateFileForWrite';
	OPCUA_BROWSENAME_GENERATESEVENT : STRING := 'GeneratesEvent';
	OPCUA_BROWSENAME_GETCERTIFICATES : STRING := 'GetCertificates';
	OPCUA_BROWSENAME_GETENCRYPTINGKEY : STRING := 'GetEncryptingKey';
	OPCUA_BROWSENAME_GETGROUPMEMBERSHIPS : STRING := 'GetGroupMemberships';
	OPCUA_BROWSENAME_GETMONITOREDITEMS : STRING := 'GetMonitoredItems';
	OPCUA_BROWSENAME_GETPOSITION : STRING := 'GetPosition';
	OPCUA_BROWSENAME_GETREJECTEDLIST : STRING := 'GetRejectedList';
	OPCUA_BROWSENAME_GETSECURITYGROUP : STRING := 'GetSecurityGroup';
	OPCUA_BROWSENAME_GETSECURITYKEYS : STRING := 'GetSecurityKeys';
	OPCUA_BROWSENAME_GROUPID : STRING := 'GroupId';
	OPCUA_BROWSENAME_GROUPPROPERTIES : STRING := 'GroupProperties';
	OPCUA_BROWSENAME_GROUPVERSION : STRING := 'GroupVersion';
	OPCUA_BROWSENAME_GUARDVARIABLETYPE : STRING := 'GuardVariableType';
	OPCUA_BROWSENAME_GUID : STRING := 'Guid';
	OPCUA_BROWSENAME_HACONFIGURATION : STRING := 'HA Configuration';
	OPCUA_BROWSENAME_HALT : STRING := 'Halt';
	OPCUA_BROWSENAME_HALTED : STRING := 'Halted';
	OPCUA_BROWSENAME_HALTEDTOREADY : STRING := 'HaltedToReady';
	OPCUA_BROWSENAME_HANDLE : STRING := 'Handle';
	OPCUA_BROWSENAME_HASADDIN : STRING := 'HasAddIn';
	OPCUA_BROWSENAME_HASALARMSUPPRESSIONGROUP : STRING := 'HasAlarmSuppressionGroup';
	OPCUA_BROWSENAME_HASARGUMENTDESCRIPTION : STRING := 'HasArgumentDescription';
	OPCUA_BROWSENAME_HASATTACHEDCOMPONENT : STRING := 'HasAttachedComponent';
	OPCUA_BROWSENAME_HASCAUSE : STRING := 'HasCause';
	OPCUA_BROWSENAME_HASCHILD : STRING := 'HasChild';
	OPCUA_BROWSENAME_HASCOMPONENT : STRING := 'HasComponent';
	OPCUA_BROWSENAME_HASCONDITION : STRING := 'HasCondition';
	OPCUA_BROWSENAME_HASCONTAINEDCOMPONENT : STRING := 'HasContainedComponent';
	OPCUA_BROWSENAME_HASDATASETREADER : STRING := 'HasDataSetReader';
	OPCUA_BROWSENAME_HASDATASETWRITER : STRING := 'HasDataSetWriter';
	OPCUA_BROWSENAME_HASDESCRIPTION : STRING := 'HasDescription';
	OPCUA_BROWSENAME_HASDICTIONARYENTRY : STRING := 'HasDictionaryEntry';
	OPCUA_BROWSENAME_HASEFFECT : STRING := 'HasEffect';
	OPCUA_BROWSENAME_HASEFFECTDISABLE : STRING := 'HasEffectDisable';
	OPCUA_BROWSENAME_HASEFFECTENABLE : STRING := 'HasEffectEnable';
	OPCUA_BROWSENAME_HASEFFECTSUPPRESSED : STRING := 'HasEffectSuppressed';
	OPCUA_BROWSENAME_HASEFFECTUNSUPPRESSED : STRING := 'HasEffectUnsuppressed';
	OPCUA_BROWSENAME_HASENCODING : STRING := 'HasEncoding';
	OPCUA_BROWSENAME_HASEVENTSOURCE : STRING := 'HasEventSource';
	OPCUA_BROWSENAME_HASFALSESUBSTATE : STRING := 'HasFalseSubState';
	OPCUA_BROWSENAME_HASGUARD : STRING := 'HasGuard';
	OPCUA_BROWSENAME_HASHISTORICALCONFIGURATION : STRING := 'HasHistoricalConfiguration';
	OPCUA_BROWSENAME_HASINTERFACE : STRING := 'HasInterface';
	OPCUA_BROWSENAME_HASLOWERLAYERINTERFACE : STRING := 'HasLowerLayerInterface';
	OPCUA_BROWSENAME_HASMODELLINGRULE : STRING := 'HasModellingRule';
	OPCUA_BROWSENAME_HASNOTIFIER : STRING := 'HasNotifier';
	OPCUA_BROWSENAME_HASOPTIONALINPUTARGUMENTDESCRIPTION : STRING := 'HasOptionalInputArgumentDescription';
	OPCUA_BROWSENAME_HASORDEREDCOMPONENT : STRING := 'HasOrderedComponent';
	OPCUA_BROWSENAME_HASPHYSICALCOMPONENT : STRING := 'HasPhysicalComponent';
	OPCUA_BROWSENAME_HASPROPERTY : STRING := 'HasProperty';
	OPCUA_BROWSENAME_HASPUBSUBCONNECTION : STRING := 'HasPubSubConnection';
	OPCUA_BROWSENAME_HASPUSHEDSECURITYGROUP : STRING := 'HasPushedSecurityGroup';
	OPCUA_BROWSENAME_HASREADERGROUP : STRING := 'HasReaderGroup';
	OPCUA_BROWSENAME_HASREFERENCEDESCRIPTION : STRING := 'HasReferenceDescription';
	OPCUA_BROWSENAME_HASSECUREELEMENT : STRING := 'HasSecureElement';
	OPCUA_BROWSENAME_HASSTRUCTUREDCOMPONENT : STRING := 'HasStructuredComponent';
	OPCUA_BROWSENAME_HASSUBSTATEMACHINE : STRING := 'HasSubStateMachine';
	OPCUA_BROWSENAME_HASSUBTYPE : STRING := 'HasSubtype';
	OPCUA_BROWSENAME_HASTRUESUBSTATE : STRING := 'HasTrueSubState';
	OPCUA_BROWSENAME_HASTYPEDEFINITION : STRING := 'HasTypeDefinition';
	OPCUA_BROWSENAME_HASWRITERGROUP : STRING := 'HasWriterGroup';
	OPCUA_BROWSENAME_HEADERLAYOUTURI : STRING := 'HeaderLayoutUri';
	OPCUA_BROWSENAME_HIERARCHICALREFERENCES : STRING := 'HierarchicalReferences';
	OPCUA_BROWSENAME_HIGH : STRING := 'High';
	OPCUA_BROWSENAME_HIGHDEADBAND : STRING := 'HighDeadband';
	OPCUA_BROWSENAME_HIGHHIGH : STRING := 'HighHigh';
	OPCUA_BROWSENAME_HIGHHIGHDEADBAND : STRING := 'HighHighDeadband';
	OPCUA_BROWSENAME_HIGHHIGHLIMIT : STRING := 'HighHighLimit';
	OPCUA_BROWSENAME_HIGHHIGHSTATE : STRING := 'HighHighState';
	OPCUA_BROWSENAME_HIGHHIGHTOHIGH : STRING := 'HighHighToHigh';
	OPCUA_BROWSENAME_HIGHLIMIT : STRING := 'HighLimit';
	OPCUA_BROWSENAME_HIGHSTATE : STRING := 'HighState';
	OPCUA_BROWSENAME_HIGHTOHIGHHIGH : STRING := 'HighToHighHigh';
	OPCUA_BROWSENAME_HIGHESTACTIVESEVERITY : STRING := 'HighestActiveSeverity';
	OPCUA_BROWSENAME_HIGHESTUNACKSEVERITY : STRING := 'HighestUnackSeverity';
	OPCUA_BROWSENAME_HIGHLYMANAGEDALARMCONDITIONCLASSTYPE : STRING := 'HighlyManagedAlarmConditionClassType';
	OPCUA_BROWSENAME_HISTORICALDATACONFIGURATIONTYPE : STRING := 'HistoricalDataConfigurationType';
	OPCUA_BROWSENAME_HISTORICALEVENTFILTER : STRING := 'HistoricalEventFilter';
	OPCUA_BROWSENAME_HISTORYEVENT : STRING := 'HistoryEvent';
	OPCUA_BROWSENAME_HISTORYEVENTFIELDLIST : STRING := 'HistoryEventFieldList';
	OPCUA_BROWSENAME_HISTORYREADCOUNT : STRING := 'HistoryReadCount';
	OPCUA_BROWSENAME_HISTORYSERVERCAPABILITIES : STRING := 'HistoryServerCapabilities';
	OPCUA_BROWSENAME_HISTORYSERVERCAPABILITIESTYPE : STRING := 'HistoryServerCapabilitiesType';
	OPCUA_BROWSENAME_HISTORYUPDATECOUNT : STRING := 'HistoryUpdateCount';
	OPCUA_BROWSENAME_HISTORYUPDATETYPE : STRING := 'HistoryUpdateType';
	OPCUA_BROWSENAME_HTTPSCERTIFICATETYPE : STRING := 'HttpsCertificateType';
	OPCUA_BROWSENAME_IBASEETHERNETCAPABILITIESTYPE : STRING := 'IBaseEthernetCapabilitiesType';
	OPCUA_BROWSENAME_IIEEEAUTONEGOTIATIONSTATUSTYPE : STRING := 'IIeeeAutoNegotiationStatusType';
	OPCUA_BROWSENAME_IIEEEBASEETHERNETPORTTYPE : STRING := 'IIeeeBaseEthernetPortType';
	OPCUA_BROWSENAME_IIEEEBASETSNSTATUSSTREAMTYPE : STRING := 'IIeeeBaseTsnStatusStreamType';
	OPCUA_BROWSENAME_IIEEEBASETSNSTREAMTYPE : STRING := 'IIeeeBaseTsnStreamType';
	OPCUA_BROWSENAME_IIEEEBASETSNTRAFFICSPECIFICATIONTYPE : STRING := 'IIeeeBaseTsnTrafficSpecificationType';
	OPCUA_BROWSENAME_IIEEETSNINTERFACECONFIGURATIONLISTENERTYPE : STRING := 'IIeeeTsnInterfaceConfigurationListenerType';
	OPCUA_BROWSENAME_IIEEETSNINTERFACECONFIGURATIONTALKERTYPE : STRING := 'IIeeeTsnInterfaceConfigurationTalkerType';
	OPCUA_BROWSENAME_IIEEETSNINTERFACECONFIGURATIONTYPE : STRING := 'IIeeeTsnInterfaceConfigurationType';
	OPCUA_BROWSENAME_IIEEETSNMACADDRESSTYPE : STRING := 'IIeeeTsnMacAddressType';
	OPCUA_BROWSENAME_IIEEETSNVLANTAGTYPE : STRING := 'IIeeeTsnVlanTagType';
	OPCUA_BROWSENAME_IIETFBASENETWORKINTERFACETYPE : STRING := 'IIetfBaseNetworkInterfaceType';
	OPCUA_BROWSENAME_IORDEREDOBJECTTYPE : STRING := 'IOrderedObjectType';
	OPCUA_BROWSENAME_IPRIORITYMAPPINGENTRYTYPE : STRING := 'IPriorityMappingEntryType';
	OPCUA_BROWSENAME_ISRCLASSTYPE : STRING := 'ISrClassType';
	OPCUA_BROWSENAME_IVLANIDTYPE : STRING := 'IVlanIdType';
	OPCUA_BROWSENAME_ICON : STRING := 'Icon';
	OPCUA_BROWSENAME_ID : STRING := 'Id';
	OPCUA_BROWSENAME_IDTYPE : STRING := 'IdType';
	OPCUA_BROWSENAME_IDENTITIES : STRING := 'Identities';
	OPCUA_BROWSENAME_IDENTITYCRITERIATYPE : STRING := 'IdentityCriteriaType';
	OPCUA_BROWSENAME_IDENTITYMAPPINGRULETYPE : STRING := 'IdentityMappingRuleType';
	OPCUA_BROWSENAME_IDLE : STRING := 'Idle';
	OPCUA_BROWSENAME_IDLETOAPPLYWRITE : STRING := 'IdleToApplyWrite';
	OPCUA_BROWSENAME_IDLETOREADPREPARE : STRING := 'IdleToReadPrepare';
	OPCUA_BROWSENAME_IETFBASENETWORKINTERFACETYPE : STRING := 'IetfBaseNetworkInterfaceType';
	OPCUA_BROWSENAME_IMAGE : STRING := 'Image';
	OPCUA_BROWSENAME_IMAGEBMP : STRING := 'ImageBMP';
	OPCUA_BROWSENAME_IMAGEGIF : STRING := 'ImageGIF';
	OPCUA_BROWSENAME_IMAGEITEMTYPE : STRING := 'ImageItemType';
	OPCUA_BROWSENAME_IMAGEJPG : STRING := 'ImageJPG';
	OPCUA_BROWSENAME_IMAGEPNG : STRING := 'ImagePNG';
	OPCUA_BROWSENAME_INDEX : STRING := 'Index';
	OPCUA_BROWSENAME_INDEXRANGE : STRING := 'IndexRange';
	OPCUA_BROWSENAME_INITIALSTATETYPE : STRING := 'InitialStateType';
	OPCUA_BROWSENAME_INPUTARGUMENTS : STRING := 'InputArguments';
	OPCUA_BROWSENAME_INPUTNODE : STRING := 'InputNode';
	OPCUA_BROWSENAME_INSERTANNOTATIONCAPABILITY : STRING := 'InsertAnnotationCapability';
	OPCUA_BROWSENAME_INSERTDATACAPABILITY : STRING := 'InsertDataCapability';
	OPCUA_BROWSENAME_INSERTEVENTCAPABILITY : STRING := 'InsertEventCapability';
	OPCUA_BROWSENAME_INSTANCECOUNT : STRING := 'InstanceCount';
	OPCUA_BROWSENAME_INSTRUMENTDIAGNOSTICALARMTYPE : STRING := 'InstrumentDiagnosticAlarmType';
	OPCUA_BROWSENAME_INSTRUMENTRANGE : STRING := 'InstrumentRange';
	OPCUA_BROWSENAME_INT16 : STRING := 'Int16';
	OPCUA_BROWSENAME_INT32 : STRING := 'Int32';
	OPCUA_BROWSENAME_INT64 : STRING := 'Int64';
	OPCUA_BROWSENAME_INTEGER : STRING := 'Integer';
	OPCUA_BROWSENAME_INTEGERID : STRING := 'IntegerId';
	OPCUA_BROWSENAME_INTERFACEADMINSTATUS : STRING := 'InterfaceAdminStatus';
	OPCUA_BROWSENAME_INTERFACENAME : STRING := 'InterfaceName';
	OPCUA_BROWSENAME_PLACEHOLDER_INTERFACENAME : STRING := '<InterfaceName>';
	OPCUA_BROWSENAME_INTERFACEOPERSTATUS : STRING := 'InterfaceOperStatus';
	OPCUA_BROWSENAME_INTERFACETYPES : STRING := 'InterfaceTypes';
	OPCUA_BROWSENAME_INTERMEDIATERESULT : STRING := 'IntermediateResult';
	OPCUA_BROWSENAME_INTERPOLATIVE : STRING := 'Interpolative';
	OPCUA_BROWSENAME_INTERVAL : STRING := 'Interval';
	OPCUA_BROWSENAME_INVALIDHOSTNAME : STRING := 'InvalidHostname';
	OPCUA_BROWSENAME_INVALIDURI : STRING := 'InvalidUri';
	OPCUA_BROWSENAME_INVALIDATEKEYS : STRING := 'InvalidateKeys';
	OPCUA_BROWSENAME_INVOCATIONCREATIONTIME : STRING := 'InvocationCreationTime';
	OPCUA_BROWSENAME_IRDIDICTIONARYENTRYTYPE : STRING := 'IrdiDictionaryEntryType';
	OPCUA_BROWSENAME_ISCONNECTED : STRING := 'IsConnected';
	OPCUA_BROWSENAME_ISDELETEMODIFIED : STRING := 'IsDeleteModified';
	OPCUA_BROWSENAME_ISDEPRECATED : STRING := 'IsDeprecated';
	OPCUA_BROWSENAME_ISEXECUTABLEON : STRING := 'IsExecutableOn';
	OPCUA_BROWSENAME_ISEXECUTINGON : STRING := 'IsExecutingOn';
	OPCUA_BROWSENAME_ISHOSTEDBY : STRING := 'IsHostedBy';
	OPCUA_BROWSENAME_ISNAMESPACESUBSET : STRING := 'IsNamespaceSubset';
	OPCUA_BROWSENAME_ISPHYSICALLYCONNECTEDTO : STRING := 'IsPhysicallyConnectedTo';
	OPCUA_BROWSENAME_ISSINGLETON : STRING := 'IsSingleton';
	OPCUA_BROWSENAME_ISSUEDIDENTITYTOKEN : STRING := 'IssuedIdentityToken';
	OPCUA_BROWSENAME_ISSUERENDPOINTURL : STRING := 'IssuerEndpointUrl';
	OPCUA_BROWSENAME_JSONDATASETMESSAGECONTENTMASK : STRING := 'JsonDataSetMessageContentMask';
	OPCUA_BROWSENAME_JSONDATASETREADERMESSAGEDATATYPE : STRING := 'JsonDataSetReaderMessageDataType';
	OPCUA_BROWSENAME_JSONDATASETREADERMESSAGETYPE : STRING := 'JsonDataSetReaderMessageType';
	OPCUA_BROWSENAME_JSONDATASETWRITERMESSAGEDATATYPE : STRING := 'JsonDataSetWriterMessageDataType';
	OPCUA_BROWSENAME_JSONDATASETWRITERMESSAGETYPE : STRING := 'JsonDataSetWriterMessageType';
	OPCUA_BROWSENAME_JSONNETWORKMESSAGECONTENTMASK : STRING := 'JsonNetworkMessageContentMask';
	OPCUA_BROWSENAME_JSONWRITERGROUPMESSAGEDATATYPE : STRING := 'JsonWriterGroupMessageDataType';
	OPCUA_BROWSENAME_JSONWRITERGROUPMESSAGETYPE : STRING := 'JsonWriterGroupMessageType';
	OPCUA_BROWSENAME_KEEPALIVETIME : STRING := 'KeepAliveTime';
	OPCUA_BROWSENAME_KEYCREDENTIALAUDITEVENTTYPE : STRING := 'KeyCredentialAuditEventType';
	OPCUA_BROWSENAME_KEYCREDENTIALCONFIGURATION : STRING := 'KeyCredentialConfiguration';
	OPCUA_BROWSENAME_KEYCREDENTIALCONFIGURATIONFOLDERTYPE : STRING := 'KeyCredentialConfigurationFolderType';
	OPCUA_BROWSENAME_KEYCREDENTIALCONFIGURATIONTYPE : STRING := 'KeyCredentialConfigurationType';
	OPCUA_BROWSENAME_KEYCREDENTIALDELETEDAUDITEVENTTYPE : STRING := 'KeyCredentialDeletedAuditEventType';
	OPCUA_BROWSENAME_KEYCREDENTIALUPDATEDAUDITEVENTTYPE : STRING := 'KeyCredentialUpdatedAuditEventType';
	OPCUA_BROWSENAME_KEYFRAMECOUNT : STRING := 'KeyFrameCount';
	OPCUA_BROWSENAME_KEYLIFETIME : STRING := 'KeyLifetime';
	OPCUA_BROWSENAME_KEYPUSHTARGETS : STRING := 'KeyPushTargets';
	OPCUA_BROWSENAME_KEYVALUEPAIR : STRING := 'KeyValuePair';
	OPCUA_BROWSENAME_LASTMETHODCALL : STRING := 'LastMethodCall';
	OPCUA_BROWSENAME_LASTMETHODCALLTIME : STRING := 'LastMethodCallTime';
	OPCUA_BROWSENAME_LASTMETHODINPUTARGUMENTS : STRING := 'LastMethodInputArguments';
	OPCUA_BROWSENAME_LASTMETHODINPUTVALUES : STRING := 'LastMethodInputValues';
	OPCUA_BROWSENAME_LASTMETHODOUTPUTARGUMENTS : STRING := 'LastMethodOutputArguments';
	OPCUA_BROWSENAME_LASTMETHODOUTPUTVALUES : STRING := 'LastMethodOutputValues';
	OPCUA_BROWSENAME_LASTMETHODRETURNSTATUS : STRING := 'LastMethodReturnStatus';
	OPCUA_BROWSENAME_LASTMETHODSESSIONID : STRING := 'LastMethodSessionId';
	OPCUA_BROWSENAME_LASTMODIFIEDTIME : STRING := 'LastModifiedTime';
	OPCUA_BROWSENAME_LASTPUSHERRORTIME : STRING := 'LastPushErrorTime';
	OPCUA_BROWSENAME_LASTPUSHEXECUTIONTIME : STRING := 'LastPushExecutionTime';
	OPCUA_BROWSENAME_LASTRESPONSE : STRING := 'LastResponse';
	OPCUA_BROWSENAME_LASTSEVERITY : STRING := 'LastSeverity';
	OPCUA_BROWSENAME_LASTTRANSITION : STRING := 'LastTransition';
	OPCUA_BROWSENAME_LASTTRANSITIONTIME : STRING := 'LastTransitionTime';
	OPCUA_BROWSENAME_LASTUPDATETIME : STRING := 'LastUpdateTime';
	OPCUA_BROWSENAME_LATCHEDSTATE : STRING := 'LatchedState';
	OPCUA_BROWSENAME_LATEPUBLISHREQUESTCOUNT : STRING := 'LatePublishRequestCount';
	OPCUA_BROWSENAME_LENGTHUNIT : STRING := 'LengthUnit';
	OPCUA_BROWSENAME_LIMITALARMTYPE : STRING := 'LimitAlarmType';
	OPCUA_BROWSENAME_LIMITSTATE : STRING := 'LimitState';
	OPCUA_BROWSENAME_LISTID : STRING := 'ListId';
	OPCUA_BROWSENAME_LISTENERSTATUS : STRING := 'ListenerStatus';
	OPCUA_BROWSENAME_LISTENERSTREAMS : STRING := 'ListenerStreams';
	OPCUA_BROWSENAME_LITERALOPERAND : STRING := 'LiteralOperand';
	OPCUA_BROWSENAME_LIVEVALUES : STRING := 'LiveValues';
	OPCUA_BROWSENAME_LOCALTIME : STRING := 'LocalTime';
	OPCUA_BROWSENAME_LOCALEID : STRING := 'LocaleId';
	OPCUA_BROWSENAME_LOCALEIDARRAY : STRING := 'LocaleIdArray';
	OPCUA_BROWSENAME_LOCALEIDS : STRING := 'LocaleIds';
	OPCUA_BROWSENAME_LOCALIZEDTEXT : STRING := 'LocalizedText';
	OPCUA_BROWSENAME_LOCATIONS : STRING := 'Locations';
	OPCUA_BROWSENAME_LOW : STRING := 'Low';
	OPCUA_BROWSENAME_LOWDEADBAND : STRING := 'LowDeadband';
	OPCUA_BROWSENAME_LOWLIMIT : STRING := 'LowLimit';
	OPCUA_BROWSENAME_LOWLOW : STRING := 'LowLow';
	OPCUA_BROWSENAME_LOWLOWDEADBAND : STRING := 'LowLowDeadband';
	OPCUA_BROWSENAME_LOWLOWLIMIT : STRING := 'LowLowLimit';
	OPCUA_BROWSENAME_LOWLOWSTATE : STRING := 'LowLowState';
	OPCUA_BROWSENAME_LOWLOWTOLOW : STRING := 'LowLowToLow';
	OPCUA_BROWSENAME_LOWSTATE : STRING := 'LowState';
	OPCUA_BROWSENAME_LOWTOLOWLOW : STRING := 'LowToLowLow';
	OPCUA_BROWSENAME_MACADDRESS : STRING := 'MacAddress';
	OPCUA_BROWSENAME_MAINTENANCECONDITIONCLASSTYPE : STRING := 'MaintenanceConditionClassType';
	OPCUA_BROWSENAME_MAJORVERSION : STRING := 'MajorVersion';
	OPCUA_BROWSENAME_MANDATORY : STRING := 'Mandatory';
	OPCUA_BROWSENAME_MANDATORYPLACEHOLDER : STRING := 'MandatoryPlaceholder';
	OPCUA_BROWSENAME_MANUFACTURERNAME : STRING := 'ManufacturerName';
	OPCUA_BROWSENAME_MAPPINGTABLES : STRING := 'MappingTables';
	OPCUA_BROWSENAME_MAPPINGURI : STRING := 'MappingUri';
	OPCUA_BROWSENAME_MAXARRAYLENGTH : STRING := 'MaxArrayLength';
	OPCUA_BROWSENAME_MAXBROWSECONTINUATIONPOINTS : STRING := 'MaxBrowseContinuationPoints';
	OPCUA_BROWSENAME_MAXBYTESTRINGLENGTH : STRING := 'MaxByteStringLength';
	OPCUA_BROWSENAME_MAXCHARACTERS : STRING := 'MaxCharacters';
	OPCUA_BROWSENAME_MAXDATASETREADERS : STRING := 'MaxDataSetReaders';
	OPCUA_BROWSENAME_MAXDATASETWRITERS : STRING := 'MaxDataSetWriters';
	OPCUA_BROWSENAME_MAXDATASETWRITERSPERGROUP : STRING := 'MaxDataSetWritersPerGroup';
	OPCUA_BROWSENAME_MAXFIELDSPERDATASET : STRING := 'MaxFieldsPerDataSet';
	OPCUA_BROWSENAME_MAXFRAMELENGTH : STRING := 'MaxFrameLength';
	OPCUA_BROWSENAME_MAXFRAMESIZE : STRING := 'MaxFrameSize';
	OPCUA_BROWSENAME_MAXFUTUREKEYCOUNT : STRING := 'MaxFutureKeyCount';
	OPCUA_BROWSENAME_MAXHISTORYCONTINUATIONPOINTS : STRING := 'MaxHistoryContinuationPoints';
	OPCUA_BROWSENAME_MAXINSTANCECOUNT : STRING := 'MaxInstanceCount';
	OPCUA_BROWSENAME_MAXINTERVALFRAMES : STRING := 'MaxIntervalFrames';
	OPCUA_BROWSENAME_MAXKEEPALIVECOUNT : STRING := 'MaxKeepAliveCount';
	OPCUA_BROWSENAME_MAXLIFETIMECOUNT : STRING := 'MaxLifetimeCount';
	OPCUA_BROWSENAME_MAXMONITOREDITEMS : STRING := 'MaxMonitoredItems';
	OPCUA_BROWSENAME_MAXMONITOREDITEMSPERCALL : STRING := 'MaxMonitoredItemsPerCall';
	OPCUA_BROWSENAME_MAXMONITOREDITEMSPERSUBSCRIPTION : STRING := 'MaxMonitoredItemsPerSubscription';
	OPCUA_BROWSENAME_MAXMONITOREDITEMSQUEUESIZE : STRING := 'MaxMonitoredItemsQueueSize';
	OPCUA_BROWSENAME_MAXNETWORKMESSAGESIZE : STRING := 'MaxNetworkMessageSize';
	OPCUA_BROWSENAME_MAXNETWORKMESSAGESIZEBROKER : STRING := 'MaxNetworkMessageSizeBroker';
	OPCUA_BROWSENAME_MAXNETWORKMESSAGESIZEDATAGRAM : STRING := 'MaxNetworkMessageSizeDatagram';
	OPCUA_BROWSENAME_MAXNODESPERBROWSE : STRING := 'MaxNodesPerBrowse';
	OPCUA_BROWSENAME_MAXNODESPERHISTORYREADDATA : STRING := 'MaxNodesPerHistoryReadData';
	OPCUA_BROWSENAME_MAXNODESPERHISTORYREADEVENTS : STRING := 'MaxNodesPerHistoryReadEvents';
	OPCUA_BROWSENAME_MAXNODESPERHISTORYUPDATEDATA : STRING := 'MaxNodesPerHistoryUpdateData';
	OPCUA_BROWSENAME_MAXNODESPERHISTORYUPDATEEVENTS : STRING := 'MaxNodesPerHistoryUpdateEvents';
	OPCUA_BROWSENAME_MAXNODESPERMETHODCALL : STRING := 'MaxNodesPerMethodCall';
	OPCUA_BROWSENAME_MAXNODESPERNODEMANAGEMENT : STRING := 'MaxNodesPerNodeManagement';
	OPCUA_BROWSENAME_MAXNODESPERREAD : STRING := 'MaxNodesPerRead';
	OPCUA_BROWSENAME_MAXNODESPERREGISTERNODES : STRING := 'MaxNodesPerRegisterNodes';
	OPCUA_BROWSENAME_MAXNODESPERTRANSLATEBROWSEPATHSTONODEIDS : STRING := 'MaxNodesPerTranslateBrowsePathsToNodeIds';
	OPCUA_BROWSENAME_MAXNODESPERWRITE : STRING := 'MaxNodesPerWrite';
	OPCUA_BROWSENAME_MAXNOTIFICATIONSPERPUBLISH : STRING := 'MaxNotificationsPerPublish';
	OPCUA_BROWSENAME_MAXPASTKEYCOUNT : STRING := 'MaxPastKeyCount';
	OPCUA_BROWSENAME_MAXPUBSUBCONNECTIONS : STRING := 'MaxPubSubConnections';
	OPCUA_BROWSENAME_MAXQUERYCONTINUATIONPOINTS : STRING := 'MaxQueryContinuationPoints';
	OPCUA_BROWSENAME_MAXREADERGROUPS : STRING := 'MaxReaderGroups';
	OPCUA_BROWSENAME_MAXRECYCLECOUNT : STRING := 'MaxRecycleCount';
	OPCUA_BROWSENAME_MAXRESPONSEMESSAGESIZE : STRING := 'MaxResponseMessageSize';
	OPCUA_BROWSENAME_MAXRETURNDATAVALUES : STRING := 'MaxReturnDataValues';
	OPCUA_BROWSENAME_MAXRETURNEVENTVALUES : STRING := 'MaxReturnEventValues';
	OPCUA_BROWSENAME_MAXSAMPLEDMONITOREDITEMSCOUNT : STRING := 'MaxSampledMonitoredItemsCount';
	OPCUA_BROWSENAME_MAXSELECTCLAUSEPARAMETERS : STRING := 'MaxSelectClauseParameters';
	OPCUA_BROWSENAME_MAXSESSIONS : STRING := 'MaxSessions';
	OPCUA_BROWSENAME_MAXSTRINGLENGTH : STRING := 'MaxStringLength';
	OPCUA_BROWSENAME_MAXSUBSCRIPTIONS : STRING := 'MaxSubscriptions';
	OPCUA_BROWSENAME_MAXSUBSCRIPTIONSPERSESSION : STRING := 'MaxSubscriptionsPerSession';
	OPCUA_BROWSENAME_MAXTIMEINTERVAL : STRING := 'MaxTimeInterval';
	OPCUA_BROWSENAME_MAXTIMESHELVED : STRING := 'MaxTimeShelved';
	OPCUA_BROWSENAME_MAXTRUSTLISTSIZE : STRING := 'MaxTrustListSize';
	OPCUA_BROWSENAME_MAXWHERECLAUSEPARAMETERS : STRING := 'MaxWhereClauseParameters';
	OPCUA_BROWSENAME_MAXWRITERGROUPS : STRING := 'MaxWriterGroups';
	OPCUA_BROWSENAME_MAXIMUM : STRING := 'Maximum';
	OPCUA_BROWSENAME_MAXIMUM2 : STRING := 'Maximum2';
	OPCUA_BROWSENAME_MAXIMUMACTIVESTATE : STRING := 'MaximumActiveState';
	OPCUA_BROWSENAME_MAXIMUMACTUALTIME : STRING := 'MaximumActualTime';
	OPCUA_BROWSENAME_MAXIMUMACTUALTIME2 : STRING := 'MaximumActualTime2';
	OPCUA_BROWSENAME_MAXIMUMALARMRATE : STRING := 'MaximumAlarmRate';
	OPCUA_BROWSENAME_MAXIMUMREALARMCOUNT : STRING := 'MaximumReAlarmCount';
	OPCUA_BROWSENAME_MAXIMUMUNACK : STRING := 'MaximumUnAck';
	OPCUA_BROWSENAME_MDNSDISCOVERYCONFIGURATION : STRING := 'MdnsDiscoveryConfiguration';
	OPCUA_BROWSENAME_MESSAGE : STRING := 'Message';
	OPCUA_BROWSENAME_MESSAGERECEIVETIMEOUT : STRING := 'MessageReceiveTimeout';
	OPCUA_BROWSENAME_MESSAGEREPEATCOUNT : STRING := 'MessageRepeatCount';
	OPCUA_BROWSENAME_MESSAGEREPEATDELAY : STRING := 'MessageRepeatDelay';
	OPCUA_BROWSENAME_MESSAGESECURITYMODE : STRING := 'MessageSecurityMode';
	OPCUA_BROWSENAME_MESSAGESEQUENCENUMBER : STRING := 'MessageSequenceNumber';
	OPCUA_BROWSENAME_MESSAGESETTINGS : STRING := 'MessageSettings';
	OPCUA_BROWSENAME_METADATAQUEUENAME : STRING := 'MetaDataQueueName';
	OPCUA_BROWSENAME_METADATAUPDATETIME : STRING := 'MetaDataUpdateTime';
	OPCUA_BROWSENAME_METHODID : STRING := 'MethodId';
	OPCUA_BROWSENAME_MIMETYPE : STRING := 'MimeType';
	OPCUA_BROWSENAME_MINSUPPORTEDSAMPLERATE : STRING := 'MinSupportedSampleRate';
	OPCUA_BROWSENAME_MINTIMEINTERVAL : STRING := 'MinTimeInterval';
	OPCUA_BROWSENAME_MINIMUM : STRING := 'Minimum';
	OPCUA_BROWSENAME_MINIMUM2 : STRING := 'Minimum2';
	OPCUA_BROWSENAME_MINIMUMACTUALTIME : STRING := 'MinimumActualTime';
	OPCUA_BROWSENAME_MINIMUMACTUALTIME2 : STRING := 'MinimumActualTime2';
	OPCUA_BROWSENAME_MINORVERSION : STRING := 'MinorVersion';
	OPCUA_BROWSENAME_MODELCHANGESTRUCTUREDATATYPE : STRING := 'ModelChangeStructureDataType';
	OPCUA_BROWSENAME_MODELLINGRULETYPE : STRING := 'ModellingRuleType';
	OPCUA_BROWSENAME_MODELLINGRULES : STRING := 'ModellingRules';
	OPCUA_BROWSENAME_MODIFYCOUNT : STRING := 'ModifyCount';
	OPCUA_BROWSENAME_MODIFYFIELDSELECTION : STRING := 'ModifyFieldSelection';
	OPCUA_BROWSENAME_MODIFYMONITOREDITEMSCOUNT : STRING := 'ModifyMonitoredItemsCount';
	OPCUA_BROWSENAME_MODIFYSUBSCRIPTIONCOUNT : STRING := 'ModifySubscriptionCount';
	OPCUA_BROWSENAME_MODIFYUSER : STRING := 'ModifyUser';
	OPCUA_BROWSENAME_MONITOREDITEMCOUNT : STRING := 'MonitoredItemCount';
	OPCUA_BROWSENAME_MONITORINGFILTER : STRING := 'MonitoringFilter';
	OPCUA_BROWSENAME_MONITORINGQUEUEOVERFLOWCOUNT : STRING := 'MonitoringQueueOverflowCount';
	OPCUA_BROWSENAME_MOVEORCOPY : STRING := 'MoveOrCopy';
	OPCUA_BROWSENAME_MULTISTATEDICTIONARYENTRYDISCRETEBASETYPE : STRING := 'MultiStateDictionaryEntryDiscreteBaseType';
	OPCUA_BROWSENAME_MULTISTATEDICTIONARYENTRYDISCRETETYPE : STRING := 'MultiStateDictionaryEntryDiscreteType';
	OPCUA_BROWSENAME_MULTISTATEDISCRETETYPE : STRING := 'MultiStateDiscreteType';
	OPCUA_BROWSENAME_MULTISTATEVALUEDISCRETETYPE : STRING := 'MultiStateValueDiscreteType';
	OPCUA_BROWSENAME_MULTICASTDNSENABLED : STRING := 'MulticastDnsEnabled';
	OPCUA_BROWSENAME_NDIMENSIONARRAYITEMTYPE : STRING := 'NDimensionArrayItemType';
	OPCUA_BROWSENAME_NAME : STRING := 'Name';
	OPCUA_BROWSENAME_NAMESPACEARRAY : STRING := 'NamespaceArray';
	OPCUA_BROWSENAME_NAMESPACEFILE : STRING := 'NamespaceFile';
	OPCUA_BROWSENAME_PLACEHOLDER_NAMESPACEIDENTIFIER : STRING := '<NamespaceIdentifier>';
	OPCUA_BROWSENAME_NAMESPACEMETADATATYPE : STRING := 'NamespaceMetadataType';
	OPCUA_BROWSENAME_NAMESPACEPUBLICATIONDATE : STRING := 'NamespacePublicationDate';
	OPCUA_BROWSENAME_NAMESPACEURI : STRING := 'NamespaceUri';
	OPCUA_BROWSENAME_NAMESPACEVERSION : STRING := 'NamespaceVersion';
	OPCUA_BROWSENAME_NAMESPACES : STRING := 'Namespaces';
	OPCUA_BROWSENAME_NAMESPACESTYPE : STRING := 'NamespacesType';
	OPCUA_BROWSENAME_NAMINGRULETYPE : STRING := 'NamingRuleType';
	OPCUA_BROWSENAME_NEGOTIATIONSTATUS : STRING := 'NegotiationStatus';
	OPCUA_BROWSENAME_NETWORKADDRESSDATATYPE : STRING := 'NetworkAddressDataType';
	OPCUA_BROWSENAME_NETWORKADDRESSTYPE : STRING := 'NetworkAddressType';
	OPCUA_BROWSENAME_NETWORKADDRESSURLDATATYPE : STRING := 'NetworkAddressUrlDataType';
	OPCUA_BROWSENAME_NETWORKADDRESSURLTYPE : STRING := 'NetworkAddressUrlType';
	OPCUA_BROWSENAME_NETWORKGROUPDATATYPE : STRING := 'NetworkGroupDataType';
	OPCUA_BROWSENAME_NETWORKINTERFACE : STRING := 'NetworkInterface';
	OPCUA_BROWSENAME_NETWORKINTERFACES : STRING := 'NetworkInterfaces';
	OPCUA_BROWSENAME_NETWORKMESSAGECONTENTMASK : STRING := 'NetworkMessageContentMask';
	OPCUA_BROWSENAME_NETWORKMESSAGENUMBER : STRING := 'NetworkMessageNumber';
	OPCUA_BROWSENAME_NEWSTATEID : STRING := 'NewStateId';
	OPCUA_BROWSENAME_NEWVALUE : STRING := 'NewValue';
	OPCUA_BROWSENAME_NEWVALUES : STRING := 'NewValues';
	OPCUA_BROWSENAME_NEXTSEQUENCENUMBER : STRING := 'NextSequenceNumber';
	OPCUA_BROWSENAME_NODEATTRIBUTESMASK : STRING := 'NodeAttributesMask';
	OPCUA_BROWSENAME_NODECLASS : STRING := 'NodeClass';
	OPCUA_BROWSENAME_NODEID : STRING := 'NodeId';
	OPCUA_BROWSENAME_NODEVERSION : STRING := 'NodeVersion';
	OPCUA_BROWSENAME_NODESTOADD : STRING := 'NodesToAdd';
	OPCUA_BROWSENAME_NODESTODELETE : STRING := 'NodesToDelete';
	OPCUA_BROWSENAME_NONEXCLUSIVEDEVIATIONALARMTYPE : STRING := 'NonExclusiveDeviationAlarmType';
	OPCUA_BROWSENAME_NONEXCLUSIVELEVELALARMTYPE : STRING := 'NonExclusiveLevelAlarmType';
	OPCUA_BROWSENAME_NONEXCLUSIVELIMITALARMTYPE : STRING := 'NonExclusiveLimitAlarmType';
	OPCUA_BROWSENAME_NONEXCLUSIVERATEOFCHANGEALARMTYPE : STRING := 'NonExclusiveRateOfChangeAlarmType';
	OPCUA_BROWSENAME_NONHIERARCHICALREFERENCES : STRING := 'NonHierarchicalReferences';
	OPCUA_BROWSENAME_NONTRANSPARENTNETWORKREDUNDANCYTYPE : STRING := 'NonTransparentNetworkRedundancyType';
	OPCUA_BROWSENAME_NONTRANSPARENTREDUNDANCYTYPE : STRING := 'NonTransparentRedundancyType';
	OPCUA_BROWSENAME_NORMALSTATE : STRING := 'NormalState';
	OPCUA_BROWSENAME_NORMALIZEDSTRING : STRING := 'NormalizedString';
	OPCUA_BROWSENAME_NOTIFICATIONSCOUNT : STRING := 'NotificationsCount';
	OPCUA_BROWSENAME_NUMBER : STRING := 'Number';
	OPCUA_BROWSENAME_NUMBERINLIST : STRING := 'NumberInList';
	OPCUA_BROWSENAME_NUMBEROFTRANSITIONS : STRING := 'NumberOfTransitions';
	OPCUA_BROWSENAME_NUMERATOR : STRING := 'Numerator';
	OPCUA_BROWSENAME_NUMERICRANGE : STRING := 'NumericRange';
	OPCUA_BROWSENAME_OPCBINARY : STRING := 'OPC Binary';
	OPCUA_BROWSENAME_OBJECTID : STRING := 'ObjectId';
	OPCUA_BROWSENAME_OBJECTTYPES : STRING := 'ObjectTypes';
	OPCUA_BROWSENAME_OBJECTS : STRING := 'Objects';
	OPCUA_BROWSENAME_OBSERVER : STRING := 'Observer';
	OPCUA_BROWSENAME_OFFDELAY : STRING := 'OffDelay';
	OPCUA_BROWSENAME_OFFNORMALALARMTYPE : STRING := 'OffNormalAlarmType';
	OPCUA_BROWSENAME_OKRESPONSE : STRING := 'OkResponse';
	OPCUA_BROWSENAME_OLDSTATEID : STRING := 'OldStateId';
	OPCUA_BROWSENAME_OLDVALUE : STRING := 'OldValue';
	OPCUA_BROWSENAME_OLDVALUES : STRING := 'OldValues';
	OPCUA_BROWSENAME_ONDELAY : STRING := 'OnDelay';
	OPCUA_BROWSENAME_ONESHOTSHELVE : STRING := 'OneShotShelve';
	OPCUA_BROWSENAME_ONESHOTSHELVE2 : STRING := 'OneShotShelve2';
	OPCUA_BROWSENAME_ONESHOTSHELVED : STRING := 'OneShotShelved';
	OPCUA_BROWSENAME_ONESHOTSHELVEDTOTIMEDSHELVED : STRING := 'OneShotShelvedToTimedShelved';
	OPCUA_BROWSENAME_ONESHOTSHELVEDTOUNSHELVED : STRING := 'OneShotShelvedToUnshelved';
	OPCUA_BROWSENAME_OPC_UA : STRING := 'Opc.Ua';
	OPCUA_BROWSENAME_OPEN : STRING := 'Open';
	OPCUA_BROWSENAME_OPENCOUNT : STRING := 'OpenCount';
	OPCUA_BROWSENAME_OPENFILEMODE : STRING := 'OpenFileMode';
	OPCUA_BROWSENAME_OPENWITHMASKS : STRING := 'OpenWithMasks';
	OPCUA_BROWSENAME_OPERSTATUS : STRING := 'OperStatus';
	OPCUA_BROWSENAME_OPERATIONLIMITS : STRING := 'OperationLimits';
	OPCUA_BROWSENAME_OPERATIONLIMITSTYPE : STRING := 'OperationLimitsType';
	OPCUA_BROWSENAME_OPERATIONALDATASETREADERS : STRING := 'OperationalDataSetReaders';
	OPCUA_BROWSENAME_OPERATIONALDATASETWRITERS : STRING := 'OperationalDataSetWriters';
	OPCUA_BROWSENAME_OPERATOR : STRING := 'Operator';
	OPCUA_BROWSENAME_OPTIONSET : STRING := 'OptionSet';
	OPCUA_BROWSENAME_OPTIONSETLENGTH : STRING := 'OptionSetLength';
	OPCUA_BROWSENAME_OPTIONSETTYPE : STRING := 'OptionSetType';
	OPCUA_BROWSENAME_OPTIONSETVALUES : STRING := 'OptionSetValues';
	OPCUA_BROWSENAME_OPTIONAL : STRING := 'Optional';
	OPCUA_BROWSENAME_OPTIONALPLACEHOLDER : STRING := 'OptionalPlaceholder';
	OPCUA_BROWSENAME_ORDEREDLISTTYPE : STRING := 'OrderedListType';
	OPCUA_BROWSENAME_PLACEHOLDER_ORDEREDOBJECT : STRING := '<OrderedObject>';
	OPCUA_BROWSENAME_ORGANIZES : STRING := 'Organizes';
	OPCUA_BROWSENAME_ORIENTATION : STRING := 'Orientation';
	OPCUA_BROWSENAME_ORIENTATIONTYPE : STRING := 'OrientationType';
	OPCUA_BROWSENAME_OUTOFSERVICESTATE : STRING := 'OutOfServiceState';
	OPCUA_BROWSENAME_OUTPUTARGUMENTS : STRING := 'OutputArguments';
	OPCUA_BROWSENAME_OVERRIDEVALUEHANDLING : STRING := 'OverrideValueHandling';
	OPCUA_BROWSENAME_PARAMETERDATATYPEID : STRING := 'ParameterDataTypeId';
	OPCUA_BROWSENAME_PASSWORDLENGTH : STRING := 'PasswordLength';
	OPCUA_BROWSENAME_PASSWORDOPTIONS : STRING := 'PasswordOptions';
	OPCUA_BROWSENAME_PASSWORDOPTIONSMASK : STRING := 'PasswordOptionsMask';
	OPCUA_BROWSENAME_PASSWORDRESTRICTIONS : STRING := 'PasswordRestrictions';
	OPCUA_BROWSENAME_PERCENTBAD : STRING := 'PercentBad';
	OPCUA_BROWSENAME_PERCENTDATABAD : STRING := 'PercentDataBad';
	OPCUA_BROWSENAME_PERCENTDATAGOOD : STRING := 'PercentDataGood';
	OPCUA_BROWSENAME_PERCENTGOOD : STRING := 'PercentGood';
	OPCUA_BROWSENAME_PERFORMINSERTREPLACE : STRING := 'PerformInsertReplace';
	OPCUA_BROWSENAME_PERFORMUPDATETYPE : STRING := 'PerformUpdateType';
	OPCUA_BROWSENAME_PERMISSIONTYPE : STRING := 'PermissionType';
	OPCUA_BROWSENAME_PHYSADDRESS : STRING := 'PhysAddress';
	OPCUA_BROWSENAME_PLACEINSERVICE : STRING := 'PlaceInService';
	OPCUA_BROWSENAME_PLACEINSERVICE2 : STRING := 'PlaceInService2';
	OPCUA_BROWSENAME_PORTABLENODEID : STRING := 'PortableNodeId';
	OPCUA_BROWSENAME_PORTABLEQUALIFIEDNAME : STRING := 'PortableQualifiedName';
	OPCUA_BROWSENAME_PRIORITY : STRING := 'Priority';
	OPCUA_BROWSENAME_PRIORITYCODEPOINT : STRING := 'PriorityCodePoint';
	OPCUA_BROWSENAME_PRIORITYLABEL : STRING := 'PriorityLabel';
	OPCUA_BROWSENAME_PRIORITYMAPPINGENTRYTYPE : STRING := 'PriorityMappingEntryType';
	OPCUA_BROWSENAME_PRIORITYMAPPINGTABLETYPE : STRING := 'PriorityMappingTableType';
	OPCUA_BROWSENAME_PRIORITYMAPPPINGENTRIES : STRING := 'PriorityMapppingEntries';
	OPCUA_BROWSENAME_PRIORITYVALUE_DSCP : STRING := 'PriorityValue_DSCP';
	OPCUA_BROWSENAME_PRIORITYVALUE_PCP : STRING := 'PriorityValue_PCP';
	OPCUA_BROWSENAME_PROCESSCONDITIONCLASSTYPE : STRING := 'ProcessConditionClassType';
	OPCUA_BROWSENAME_PROCESSINGOFFSET : STRING := 'ProcessingOffset';
	OPCUA_BROWSENAME_PRODUCTNAME : STRING := 'ProductName';
	OPCUA_BROWSENAME_PRODUCTURI : STRING := 'ProductUri';
	OPCUA_BROWSENAME_PROFILEURI : STRING := 'ProfileUri';
	OPCUA_BROWSENAME_PROGRAMDIAGNOSTIC : STRING := 'ProgramDiagnostic';
	OPCUA_BROWSENAME_PROGRAMDIAGNOSTIC2DATATYPE : STRING := 'ProgramDiagnostic2DataType';
	OPCUA_BROWSENAME_PROGRAMDIAGNOSTIC2TYPE : STRING := 'ProgramDiagnostic2Type';
	OPCUA_BROWSENAME_PROGRAMDIAGNOSTICDATATYPE : STRING := 'ProgramDiagnosticDataType';
	OPCUA_BROWSENAME_PROGRAMDIAGNOSTICTYPE : STRING := 'ProgramDiagnosticType';
	OPCUA_BROWSENAME_PROGRAMSTATEMACHINETYPE : STRING := 'ProgramStateMachineType';
	OPCUA_BROWSENAME_PROGRAMTRANSITIONAUDITEVENTTYPE : STRING := 'ProgramTransitionAuditEventType';
	OPCUA_BROWSENAME_PROGRAMTRANSITIONEVENTTYPE : STRING := 'ProgramTransitionEventType';
	OPCUA_BROWSENAME_PROGRESS : STRING := 'Progress';
	OPCUA_BROWSENAME_PROGRESSEVENTTYPE : STRING := 'ProgressEventType';
	OPCUA_BROWSENAME_PROMPT : STRING := 'Prompt';
	OPCUA_BROWSENAME_PROPERTYTYPE : STRING := 'PropertyType';
	OPCUA_BROWSENAME_PROVISIONABLEDEVICE : STRING := 'ProvisionableDevice';
	OPCUA_BROWSENAME_PROVISIONABLEDEVICETYPE : STRING := 'ProvisionableDeviceType';
	OPCUA_BROWSENAME_PUBSUBCAPABILITIESTYPE : STRING := 'PubSubCapabilitiesType';
	OPCUA_BROWSENAME_PUBSUBCAPABLITIES : STRING := 'PubSubCapablities';
	OPCUA_BROWSENAME_PUBSUBCOMMUNICATIONFAILUREEVENTTYPE : STRING := 'PubSubCommunicationFailureEventType';
	OPCUA_BROWSENAME_PUBSUBCONFIGURATION : STRING := 'PubSubConfiguration';
	OPCUA_BROWSENAME_PUBSUBCONFIGURATION2DATATYPE : STRING := 'PubSubConfiguration2DataType';
	OPCUA_BROWSENAME_PUBSUBCONFIGURATIONDATATYPE : STRING := 'PubSubConfigurationDataType';
	OPCUA_BROWSENAME_PUBSUBCONFIGURATIONREFDATATYPE : STRING := 'PubSubConfigurationRefDataType';
	OPCUA_BROWSENAME_PUBSUBCONFIGURATIONREFMASK : STRING := 'PubSubConfigurationRefMask';
	OPCUA_BROWSENAME_PUBSUBCONFIGURATIONTYPE : STRING := 'PubSubConfigurationType';
	OPCUA_BROWSENAME_PUBSUBCONFIGURATIONVALUEDATATYPE : STRING := 'PubSubConfigurationValueDataType';
	OPCUA_BROWSENAME_PUBSUBCONNECTIONDATATYPE : STRING := 'PubSubConnectionDataType';
	OPCUA_BROWSENAME_PUBSUBCONNECTIONTYPE : STRING := 'PubSubConnectionType';
	OPCUA_BROWSENAME_PUBSUBDIAGNOSTICSCONNECTIONTYPE : STRING := 'PubSubDiagnosticsConnectionType';
	OPCUA_BROWSENAME_PUBSUBDIAGNOSTICSCOUNTERCLASSIFICATION : STRING := 'PubSubDiagnosticsCounterClassification';
	OPCUA_BROWSENAME_PUBSUBDIAGNOSTICSCOUNTERTYPE : STRING := 'PubSubDiagnosticsCounterType';
	OPCUA_BROWSENAME_PUBSUBDIAGNOSTICSDATASETREADERTYPE : STRING := 'PubSubDiagnosticsDataSetReaderType';
	OPCUA_BROWSENAME_PUBSUBDIAGNOSTICSDATASETWRITERTYPE : STRING := 'PubSubDiagnosticsDataSetWriterType';
	OPCUA_BROWSENAME_PUBSUBDIAGNOSTICSREADERGROUPTYPE : STRING := 'PubSubDiagnosticsReaderGroupType';
	OPCUA_BROWSENAME_PUBSUBDIAGNOSTICSROOTTYPE : STRING := 'PubSubDiagnosticsRootType';
	OPCUA_BROWSENAME_PUBSUBDIAGNOSTICSTYPE : STRING := 'PubSubDiagnosticsType';
	OPCUA_BROWSENAME_PUBSUBDIAGNOSTICSWRITERGROUPTYPE : STRING := 'PubSubDiagnosticsWriterGroupType';
	OPCUA_BROWSENAME_PUBSUBGROUPDATATYPE : STRING := 'PubSubGroupDataType';
	OPCUA_BROWSENAME_PUBSUBGROUPTYPE : STRING := 'PubSubGroupType';
	OPCUA_BROWSENAME_PUBSUBKEYPUSHTARGETDATATYPE : STRING := 'PubSubKeyPushTargetDataType';
	OPCUA_BROWSENAME_PUBSUBKEYPUSHTARGETFOLDERTYPE : STRING := 'PubSubKeyPushTargetFolderType';
	OPCUA_BROWSENAME_PUBSUBKEYPUSHTARGETTYPE : STRING := 'PubSubKeyPushTargetType';
	OPCUA_BROWSENAME_PUBSUBKEYSERVICETYPE : STRING := 'PubSubKeyServiceType';
	OPCUA_BROWSENAME_PUBSUBSTATE : STRING := 'PubSubState';
	OPCUA_BROWSENAME_PUBSUBSTATUSEVENTTYPE : STRING := 'PubSubStatusEventType';
	OPCUA_BROWSENAME_PUBSUBSTATUSTYPE : STRING := 'PubSubStatusType';
	OPCUA_BROWSENAME_PUBSUBTRANSPORTLIMITSEXCEEDEVENTTYPE : STRING := 'PubSubTransportLimitsExceedEventType';
	OPCUA_BROWSENAME_PUBLISHCOUNT : STRING := 'PublishCount';
	OPCUA_BROWSENAME_PUBLISHREQUESTCOUNT : STRING := 'PublishRequestCount';
	OPCUA_BROWSENAME_PUBLISHSUBSCRIBE : STRING := 'PublishSubscribe';
	OPCUA_BROWSENAME_PUBLISHSUBSCRIBETYPE : STRING := 'PublishSubscribeType';
	OPCUA_BROWSENAME_PUBLISHEDDATA : STRING := 'PublishedData';
	OPCUA_BROWSENAME_PUBLISHEDDATAITEMSDATATYPE : STRING := 'PublishedDataItemsDataType';
	OPCUA_BROWSENAME_PUBLISHEDDATAITEMSTYPE : STRING := 'PublishedDataItemsType';
	OPCUA_BROWSENAME_PUBLISHEDDATASETCUSTOMSOURCEDATATYPE : STRING := 'PublishedDataSetCustomSourceDataType';
	OPCUA_BROWSENAME_PUBLISHEDDATASETDATATYPE : STRING := 'PublishedDataSetDataType';
	OPCUA_BROWSENAME_PLACEHOLDER_PUBLISHEDDATASETNAME : STRING := '<PublishedDataSetName>';
	OPCUA_BROWSENAME_PUBLISHEDDATASETSOURCEDATATYPE : STRING := 'PublishedDataSetSourceDataType';
	OPCUA_BROWSENAME_PUBLISHEDDATASETTYPE : STRING := 'PublishedDataSetType';
	OPCUA_BROWSENAME_PUBLISHEDDATASETS : STRING := 'PublishedDataSets';
	OPCUA_BROWSENAME_PUBLISHEDEVENTSDATATYPE : STRING := 'PublishedEventsDataType';
	OPCUA_BROWSENAME_PUBLISHEDEVENTSTYPE : STRING := 'PublishedEventsType';
	OPCUA_BROWSENAME_PUBLISHEDVARIABLEDATATYPE : STRING := 'PublishedVariableDataType';
	OPCUA_BROWSENAME_PUBLISHERID : STRING := 'PublisherId';
	OPCUA_BROWSENAME_PUBLISHINGENABLED : STRING := 'PublishingEnabled';
	OPCUA_BROWSENAME_PUBLISHINGINTERVAL : STRING := 'PublishingInterval';
	OPCUA_BROWSENAME_PUBLISHINGINTERVALCOUNT : STRING := 'PublishingIntervalCount';
	OPCUA_BROWSENAME_PUBLISHINGOFFSET : STRING := 'PublishingOffset';
	OPCUA_BROWSENAME_PLACEHOLDER_PUSHTARGETFOLDERNAME : STRING := '<PushTargetFolderName>';
	OPCUA_BROWSENAME_PLACEHOLDER_PUSHTARGETNAME : STRING := '<PushTargetName>';
	OPCUA_BROWSENAME_QOSCATEGORY : STRING := 'QosCategory';
	OPCUA_BROWSENAME_QOSDATATYPE : STRING := 'QosDataType';
	OPCUA_BROWSENAME_QUALIFIEDNAME : STRING := 'QualifiedName';
	OPCUA_BROWSENAME_QUALITY : STRING := 'Quality';
	OPCUA_BROWSENAME_QUERYFIRSTCOUNT : STRING := 'QueryFirstCount';
	OPCUA_BROWSENAME_QUERYNEXTCOUNT : STRING := 'QueryNextCount';
	OPCUA_BROWSENAME_QUEUENAME : STRING := 'QueueName';
	OPCUA_BROWSENAME_RANGE : STRING := 'Range';
	OPCUA_BROWSENAME_RANGE2 : STRING := 'Range2';
	OPCUA_BROWSENAME_RATE : STRING := 'Rate';
	OPCUA_BROWSENAME_RATIONALNUMBER : STRING := 'RationalNumber';
	OPCUA_BROWSENAME_RATIONALNUMBERTYPE : STRING := 'RationalNumberType';
	OPCUA_BROWSENAME_REALARMREPEATCOUNT : STRING := 'ReAlarmRepeatCount';
	OPCUA_BROWSENAME_REALARMTIME : STRING := 'ReAlarmTime';
	OPCUA_BROWSENAME_READ : STRING := 'Read';
	OPCUA_BROWSENAME_READCOUNT : STRING := 'ReadCount';
	OPCUA_BROWSENAME_READPREPARE : STRING := 'ReadPrepare';
	OPCUA_BROWSENAME_READPREPARETOERROR : STRING := 'ReadPrepareToError';
	OPCUA_BROWSENAME_READPREPARETOREADTRANSFER : STRING := 'ReadPrepareToReadTransfer';
	OPCUA_BROWSENAME_READTRANSFER : STRING := 'ReadTransfer';
	OPCUA_BROWSENAME_READTRANSFERTOERROR : STRING := 'ReadTransferToError';
	OPCUA_BROWSENAME_READTRANSFERTOIDLE : STRING := 'ReadTransferToIdle';
	OPCUA_BROWSENAME_READERGROUPDATATYPE : STRING := 'ReaderGroupDataType';
	OPCUA_BROWSENAME_READERGROUPMESSAGEDATATYPE : STRING := 'ReaderGroupMessageDataType';
	OPCUA_BROWSENAME_READERGROUPMESSAGETYPE : STRING := 'ReaderGroupMessageType';
	OPCUA_BROWSENAME_PLACEHOLDER_READERGROUPNAME : STRING := '<ReaderGroupName>';
	OPCUA_BROWSENAME_READERGROUPTRANSPORTDATATYPE : STRING := 'ReaderGroupTransportDataType';
	OPCUA_BROWSENAME_READERGROUPTRANSPORTTYPE : STRING := 'ReaderGroupTransportType';
	OPCUA_BROWSENAME_READERGROUPTYPE : STRING := 'ReaderGroupType';
	OPCUA_BROWSENAME_READY : STRING := 'Ready';
	OPCUA_BROWSENAME_READYTOHALTED : STRING := 'ReadyToHalted';
	OPCUA_BROWSENAME_READYTORUNNING : STRING := 'ReadyToRunning';
	OPCUA_BROWSENAME_RECEIVEOFFSET : STRING := 'ReceiveOffset';
	OPCUA_BROWSENAME_RECEIVEQOSDATATYPE : STRING := 'ReceiveQosDataType';
	OPCUA_BROWSENAME_RECEIVEQOSPRIORITYDATATYPE : STRING := 'ReceiveQosPriorityDataType';
	OPCUA_BROWSENAME_RECEIVETIME : STRING := 'ReceiveTime';
	OPCUA_BROWSENAME_RECEIVEDINVALIDNETWORKMESSAGES : STRING := 'ReceivedInvalidNetworkMessages';
	OPCUA_BROWSENAME_RECEIVEDNETWORKMESSAGES : STRING := 'ReceivedNetworkMessages';
	OPCUA_BROWSENAME_RECYCLECOUNT : STRING := 'RecycleCount';
	OPCUA_BROWSENAME_REDUNDANCYSUPPORT : STRING := 'RedundancySupport';
	OPCUA_BROWSENAME_REDUNDANTSERVERARRAY : STRING := 'RedundantServerArray';
	OPCUA_BROWSENAME_REDUNDANTSERVERDATATYPE : STRING := 'RedundantServerDataType';
	OPCUA_BROWSENAME_REFERENCEDESCRIPTIONDATATYPE : STRING := 'ReferenceDescriptionDataType';
	OPCUA_BROWSENAME_REFERENCEDESCRIPTIONVARIABLETYPE : STRING := 'ReferenceDescriptionVariableType';
	OPCUA_BROWSENAME_REFERENCELISTENTRYDATATYPE : STRING := 'ReferenceListEntryDataType';
	OPCUA_BROWSENAME_REFERENCEREFINEMENT : STRING := 'ReferenceRefinement';
	OPCUA_BROWSENAME_REFERENCETYPES : STRING := 'ReferenceTypes';
	OPCUA_BROWSENAME_REFERENCES : STRING := 'References';
	OPCUA_BROWSENAME_REFERENCESTOADD : STRING := 'ReferencesToAdd';
	OPCUA_BROWSENAME_REFERENCESTODELETE : STRING := 'ReferencesToDelete';
	OPCUA_BROWSENAME_REFRESHENDEVENTTYPE : STRING := 'RefreshEndEventType';
	OPCUA_BROWSENAME_REFRESHREQUIREDEVENTTYPE : STRING := 'RefreshRequiredEventType';
	OPCUA_BROWSENAME_REFRESHSTARTEVENTTYPE : STRING := 'RefreshStartEventType';
	OPCUA_BROWSENAME_REGISTERNODESCOUNT : STRING := 'RegisterNodesCount';
	OPCUA_BROWSENAME_REGISTEREDSERVER : STRING := 'RegisteredServer';
	OPCUA_BROWSENAME_REJECTEDREQUESTSCOUNT : STRING := 'RejectedRequestsCount';
	OPCUA_BROWSENAME_REJECTEDSESSIONCOUNT : STRING := 'RejectedSessionCount';
	OPCUA_BROWSENAME_RELATIVEPATH : STRING := 'RelativePath';
	OPCUA_BROWSENAME_RELATIVEPATHELEMENT : STRING := 'RelativePathElement';
	OPCUA_BROWSENAME_REMOVEAPPLICATION : STRING := 'RemoveApplication';
	OPCUA_BROWSENAME_REMOVECERTIFICATE : STRING := 'RemoveCertificate';
	OPCUA_BROWSENAME_REMOVECONNECTION : STRING := 'RemoveConnection';
	OPCUA_BROWSENAME_REMOVEDATASETFOLDER : STRING := 'RemoveDataSetFolder';
	OPCUA_BROWSENAME_REMOVEDATASETREADER : STRING := 'RemoveDataSetReader';
	OPCUA_BROWSENAME_REMOVEDATASETWRITER : STRING := 'RemoveDataSetWriter';
	OPCUA_BROWSENAME_REMOVEENDPOINT : STRING := 'RemoveEndpoint';
	OPCUA_BROWSENAME_REMOVEEXTENSIONFIELD : STRING := 'RemoveExtensionField';
	OPCUA_BROWSENAME_REMOVEFROMSERVICE : STRING := 'RemoveFromService';
	OPCUA_BROWSENAME_REMOVEFROMSERVICE2 : STRING := 'RemoveFromService2';
	OPCUA_BROWSENAME_REMOVEGROUP : STRING := 'RemoveGroup';
	OPCUA_BROWSENAME_REMOVEIDENTITY : STRING := 'RemoveIdentity';
	OPCUA_BROWSENAME_REMOVEPUBLISHEDDATASET : STRING := 'RemovePublishedDataSet';
	OPCUA_BROWSENAME_REMOVEPUSHTARGET : STRING := 'RemovePushTarget';
	OPCUA_BROWSENAME_REMOVEPUSHTARGETFOLDER : STRING := 'RemovePushTargetFolder';
	OPCUA_BROWSENAME_REMOVEROLE : STRING := 'RemoveRole';
	OPCUA_BROWSENAME_REMOVESECURITYGROUP : STRING := 'RemoveSecurityGroup';
	OPCUA_BROWSENAME_REMOVESECURITYGROUPFOLDER : STRING := 'RemoveSecurityGroupFolder';
	OPCUA_BROWSENAME_REMOVESUBSCRIBEDDATASET : STRING := 'RemoveSubscribedDataSet';
	OPCUA_BROWSENAME_REMOVETARGETVARIABLES : STRING := 'RemoveTargetVariables';
	OPCUA_BROWSENAME_REMOVEUSER : STRING := 'RemoveUser';
	OPCUA_BROWSENAME_REMOVEVARIABLES : STRING := 'RemoveVariables';
	OPCUA_BROWSENAME_REPLACEDATACAPABILITY : STRING := 'ReplaceDataCapability';
	OPCUA_BROWSENAME_REPLACEEVENTCAPABILITY : STRING := 'ReplaceEventCapability';
	OPCUA_BROWSENAME_REPRESENTSSAMEENTITYAS : STRING := 'RepresentsSameEntityAs';
	OPCUA_BROWSENAME_REPRESENTSSAMEFUNCTIONALITYAS : STRING := 'RepresentsSameFunctionalityAs';
	OPCUA_BROWSENAME_REPRESENTSSAMEHARDWAREAS : STRING := 'RepresentsSameHardwareAs';
	OPCUA_BROWSENAME_REPUBLISHCOUNT : STRING := 'RepublishCount';
	OPCUA_BROWSENAME_REPUBLISHMESSAGECOUNT : STRING := 'RepublishMessageCount';
	OPCUA_BROWSENAME_REPUBLISHMESSAGEREQUESTCOUNT : STRING := 'RepublishMessageRequestCount';
	OPCUA_BROWSENAME_REPUBLISHREQUESTCOUNT : STRING := 'RepublishRequestCount';
	OPCUA_BROWSENAME_REQTIMES : STRING := 'ReqTimes';
	OPCUA_BROWSENAME_REQUESTHANDLE : STRING := 'RequestHandle';
	OPCUA_BROWSENAME_REQUESTSERVERSTATECHANGE : STRING := 'RequestServerStateChange';
	OPCUA_BROWSENAME_REQUESTTICKETS : STRING := 'RequestTickets';
	OPCUA_BROWSENAME_REQUESTTYPE : STRING := 'RequestType';
	OPCUA_BROWSENAME_REQUESTEDDELIVERYGUARANTEE : STRING := 'RequestedDeliveryGuarantee';
	OPCUA_BROWSENAME_REQUESTEDKEYCOUNT : STRING := 'RequestedKeyCount';
	OPCUA_BROWSENAME_REQUESTEDLIFETIME : STRING := 'RequestedLifetime';
	OPCUA_BROWSENAME_REQUIRES : STRING := 'Requires';
	OPCUA_BROWSENAME_RESENDDATA : STRING := 'ResendData';
	OPCUA_BROWSENAME_RESERVEIDS : STRING := 'ReserveIds';
	OPCUA_BROWSENAME_RESET : STRING := 'Reset';
	OPCUA_BROWSENAME_RESET2 : STRING := 'Reset2';
	OPCUA_BROWSENAME_RESETTOSERVERDEFAULTS : STRING := 'ResetToServerDefaults';
	OPCUA_BROWSENAME_RESOLVEDADDRESS : STRING := 'ResolvedAddress';
	OPCUA_BROWSENAME_RESOURCEURI : STRING := 'ResourceUri';
	OPCUA_BROWSENAME_RESOURCES : STRING := 'Resources';
	OPCUA_BROWSENAME_RESPOND : STRING := 'Respond';
	OPCUA_BROWSENAME_RESPOND2 : STRING := 'Respond2';
	OPCUA_BROWSENAME_RESPONSEOPTIONSET : STRING := 'ResponseOptionSet';
	OPCUA_BROWSENAME_RESTRICTTOLIST : STRING := 'RestrictToList';
	OPCUA_BROWSENAME_RESULT : STRING := 'Result';
	OPCUA_BROWSENAME_RESUME : STRING := 'Resume';
	OPCUA_BROWSENAME_RETAIN : STRING := 'Retain';
	OPCUA_BROWSENAME_RETRYINTERVAL : STRING := 'RetryInterval';
	OPCUA_BROWSENAME_REVISEDSESSIONTIMEOUT : STRING := 'RevisedSessionTimeout';
	OPCUA_BROWSENAME_ROLEMAPPINGRULECHANGEDAUDITEVENTTYPE : STRING := 'RoleMappingRuleChangedAuditEventType';
	OPCUA_BROWSENAME_PLACEHOLDER_ROLENAME : STRING := '<RoleName>';
	OPCUA_BROWSENAME_ROLEPERMISSIONTYPE : STRING := 'RolePermissionType';
	OPCUA_BROWSENAME_ROLESET : STRING := 'RoleSet';
	OPCUA_BROWSENAME_ROLESETTYPE : STRING := 'RoleSetType';
	OPCUA_BROWSENAME_ROLETYPE : STRING := 'RoleType';
	OPCUA_BROWSENAME_ROOT : STRING := 'Root';
	OPCUA_BROWSENAME_RSAMINAPPLICATIONCERTIFICATETYPE : STRING := 'RsaMinApplicationCertificateType';
	OPCUA_BROWSENAME_RSASHA256APPLICATIONCERTIFICATETYPE : STRING := 'RsaSha256ApplicationCertificateType';
	OPCUA_BROWSENAME_RUNNING : STRING := 'Running';
	OPCUA_BROWSENAME_RUNNINGTOHALTED : STRING := 'RunningToHalted';
	OPCUA_BROWSENAME_RUNNINGTOREADY : STRING := 'RunningToReady';
	OPCUA_BROWSENAME_RUNNINGTOSUSPENDED : STRING := 'RunningToSuspended';
	OPCUA_BROWSENAME_SBYTE : STRING := 'SByte';
	OPCUA_BROWSENAME_SAFETYCONDITIONCLASSTYPE : STRING := 'SafetyConditionClassType';
	OPCUA_BROWSENAME_SAMPLEDMONITOREDITEMSCOUNT : STRING := 'SampledMonitoredItemsCount';
	OPCUA_BROWSENAME_SAMPLINGINTERVAL : STRING := 'SamplingInterval';
	OPCUA_BROWSENAME_SAMPLINGINTERVALDIAGNOSTICS : STRING := 'SamplingIntervalDiagnostics';
	OPCUA_BROWSENAME_SAMPLINGINTERVALDIAGNOSTICSARRAY : STRING := 'SamplingIntervalDiagnosticsArray';
	OPCUA_BROWSENAME_SAMPLINGINTERVALDIAGNOSTICSARRAYTYPE : STRING := 'SamplingIntervalDiagnosticsArrayType';
	OPCUA_BROWSENAME_SAMPLINGINTERVALDIAGNOSTICSDATATYPE : STRING := 'SamplingIntervalDiagnosticsDataType';
	OPCUA_BROWSENAME_SAMPLINGINTERVALDIAGNOSTICSTYPE : STRING := 'SamplingIntervalDiagnosticsType';
	OPCUA_BROWSENAME_SAMPLINGOFFSET : STRING := 'SamplingOffset';
	OPCUA_BROWSENAME_SECONDSTILLSHUTDOWN : STRING := 'SecondsTillShutdown';
	OPCUA_BROWSENAME_SECURECHANNELID : STRING := 'SecureChannelId';
	OPCUA_BROWSENAME_SECURITYADMIN : STRING := 'SecurityAdmin';
	OPCUA_BROWSENAME_SECURITYGROUPDATATYPE : STRING := 'SecurityGroupDataType';
	OPCUA_BROWSENAME_PLACEHOLDER_SECURITYGROUPFOLDERNAME : STRING := '<SecurityGroupFolderName>';
	OPCUA_BROWSENAME_SECURITYGROUPFOLDERTYPE : STRING := 'SecurityGroupFolderType';
	OPCUA_BROWSENAME_SECURITYGROUPID : STRING := 'SecurityGroupId';
	OPCUA_BROWSENAME_PLACEHOLDER_SECURITYGROUPNAME : STRING := '<SecurityGroupName>';
	OPCUA_BROWSENAME_SECURITYGROUPTYPE : STRING := 'SecurityGroupType';
	OPCUA_BROWSENAME_SECURITYGROUPS : STRING := 'SecurityGroups';
	OPCUA_BROWSENAME_SECURITYKEYSERVERACCESS : STRING := 'SecurityKeyServerAccess';
	OPCUA_BROWSENAME_SECURITYKEYSERVERADMIN : STRING := 'SecurityKeyServerAdmin';
	OPCUA_BROWSENAME_SECURITYKEYSERVERPUSH : STRING := 'SecurityKeyServerPush';
	OPCUA_BROWSENAME_SECURITYKEYSERVICES : STRING := 'SecurityKeyServices';
	OPCUA_BROWSENAME_SECURITYMODE : STRING := 'SecurityMode';
	OPCUA_BROWSENAME_SECURITYPOLICYURI : STRING := 'SecurityPolicyUri';
	OPCUA_BROWSENAME_SECURITYREJECTEDREQUESTSCOUNT : STRING := 'SecurityRejectedRequestsCount';
	OPCUA_BROWSENAME_SECURITYREJECTEDSESSIONCOUNT : STRING := 'SecurityRejectedSessionCount';
	OPCUA_BROWSENAME_SECURITYTOKENID : STRING := 'SecurityTokenID';
	OPCUA_BROWSENAME_SECURITYTOKENREQUESTTYPE : STRING := 'SecurityTokenRequestType';
	OPCUA_BROWSENAME_SELECTEDFIELDS : STRING := 'SelectedFields';
	OPCUA_BROWSENAME_SELECTEDRESPONSE : STRING := 'SelectedResponse';
	OPCUA_BROWSENAME_SELECTIONDESCRIPTIONS : STRING := 'SelectionDescriptions';
	OPCUA_BROWSENAME_SELECTIONLISTTYPE : STRING := 'SelectionListType';
	OPCUA_BROWSENAME_SELECTIONS : STRING := 'Selections';
	OPCUA_BROWSENAME_SEMANTICCHANGEEVENTTYPE : STRING := 'SemanticChangeEventType';
	OPCUA_BROWSENAME_SEMANTICCHANGESTRUCTUREDATATYPE : STRING := 'SemanticChangeStructureDataType';
	OPCUA_BROWSENAME_SEMANTICVERSIONSTRING : STRING := 'SemanticVersionString';
	OPCUA_BROWSENAME_SENTNETWORKMESSAGES : STRING := 'SentNetworkMessages';
	OPCUA_BROWSENAME_SERVER : STRING := 'Server';
	OPCUA_BROWSENAME_SERVERARRAY : STRING := 'ServerArray';
	OPCUA_BROWSENAME_SERVERCAPABILITIES : STRING := 'ServerCapabilities';
	OPCUA_BROWSENAME_SERVERCAPABILITIESTYPE : STRING := 'ServerCapabilitiesType';
	OPCUA_BROWSENAME_SERVERCONFIGURATION : STRING := 'ServerConfiguration';
	OPCUA_BROWSENAME_SERVERCONFIGURATIONTYPE : STRING := 'ServerConfigurationType';
	OPCUA_BROWSENAME_SERVERDIAGNOSTICS : STRING := 'ServerDiagnostics';
	OPCUA_BROWSENAME_SERVERDIAGNOSTICSSUMMARY : STRING := 'ServerDiagnosticsSummary';
	OPCUA_BROWSENAME_SERVERDIAGNOSTICSSUMMARYDATATYPE : STRING := 'ServerDiagnosticsSummaryDataType';
	OPCUA_BROWSENAME_SERVERDIAGNOSTICSSUMMARYTYPE : STRING := 'ServerDiagnosticsSummaryType';
	OPCUA_BROWSENAME_SERVERDIAGNOSTICSTYPE : STRING := 'ServerDiagnosticsType';
	OPCUA_BROWSENAME_SERVERID : STRING := 'ServerId';
	OPCUA_BROWSENAME_SERVERNETWORKGROUPS : STRING := 'ServerNetworkGroups';
	OPCUA_BROWSENAME_SERVERONNETWORK : STRING := 'ServerOnNetwork';
	OPCUA_BROWSENAME_SERVERPROFILEARRAY : STRING := 'ServerProfileArray';
	OPCUA_BROWSENAME_SERVERREDUNDANCY : STRING := 'ServerRedundancy';
	OPCUA_BROWSENAME_SERVERREDUNDANCYTYPE : STRING := 'ServerRedundancyType';
	OPCUA_BROWSENAME_SERVERSTATE : STRING := 'ServerState';
	OPCUA_BROWSENAME_SERVERSTATUS : STRING := 'ServerStatus';
	OPCUA_BROWSENAME_SERVERSTATUSDATATYPE : STRING := 'ServerStatusDataType';
	OPCUA_BROWSENAME_SERVERSTATUSTYPE : STRING := 'ServerStatusType';
	OPCUA_BROWSENAME_SERVERTIMESTAMPSUPPORTED : STRING := 'ServerTimestampSupported';
	OPCUA_BROWSENAME_SERVERTYPE : STRING := 'ServerType';
	OPCUA_BROWSENAME_SERVERURI : STRING := 'ServerUri';
	OPCUA_BROWSENAME_SERVERURIARRAY : STRING := 'ServerUriArray';
	OPCUA_BROWSENAME_SERVERVENDORCAPABILITYTYPE : STRING := 'ServerVendorCapabilityType';
	OPCUA_BROWSENAME_SERVERVIEWCOUNT : STRING := 'ServerViewCount';
	OPCUA_BROWSENAME_SERVICECERTIFICATE : STRING := 'ServiceCertificate';
	OPCUA_BROWSENAME_SERVICECOUNTERDATATYPE : STRING := 'ServiceCounterDataType';
	OPCUA_BROWSENAME_SERVICELEVEL : STRING := 'ServiceLevel';
	OPCUA_BROWSENAME_PLACEHOLDER_SERVICENAME : STRING := '<ServiceName>';
	OPCUA_BROWSENAME_SERVICESTATUS : STRING := 'ServiceStatus';
	OPCUA_BROWSENAME_SERVICEURI : STRING := 'ServiceUri';
	OPCUA_BROWSENAME_SESSIONABORTCOUNT : STRING := 'SessionAbortCount';
	OPCUA_BROWSENAME_SESSIONAUTHENTICATIONTOKEN : STRING := 'SessionAuthenticationToken';
	OPCUA_BROWSENAME_SESSIONDIAGNOSTICS : STRING := 'SessionDiagnostics';
	OPCUA_BROWSENAME_SESSIONDIAGNOSTICSARRAY : STRING := 'SessionDiagnosticsArray';
	OPCUA_BROWSENAME_SESSIONDIAGNOSTICSARRAYTYPE : STRING := 'SessionDiagnosticsArrayType';
	OPCUA_BROWSENAME_SESSIONDIAGNOSTICSDATATYPE : STRING := 'SessionDiagnosticsDataType';
	OPCUA_BROWSENAME_SESSIONDIAGNOSTICSOBJECTTYPE : STRING := 'SessionDiagnosticsObjectType';
	OPCUA_BROWSENAME_SESSIONDIAGNOSTICSVARIABLETYPE : STRING := 'SessionDiagnosticsVariableType';
	OPCUA_BROWSENAME_SESSIONID : STRING := 'SessionId';
	OPCUA_BROWSENAME_SESSIONNAME : STRING := 'SessionName';
	OPCUA_BROWSENAME_SESSIONSECURITYDIAGNOSTICS : STRING := 'SessionSecurityDiagnostics';
	OPCUA_BROWSENAME_SESSIONSECURITYDIAGNOSTICSARRAY : STRING := 'SessionSecurityDiagnosticsArray';
	OPCUA_BROWSENAME_SESSIONSECURITYDIAGNOSTICSARRAYTYPE : STRING := 'SessionSecurityDiagnosticsArrayType';
	OPCUA_BROWSENAME_SESSIONSECURITYDIAGNOSTICSDATATYPE : STRING := 'SessionSecurityDiagnosticsDataType';
	OPCUA_BROWSENAME_SESSIONSECURITYDIAGNOSTICSTYPE : STRING := 'SessionSecurityDiagnosticsType';
	OPCUA_BROWSENAME_SESSIONTIMEOUTCOUNT : STRING := 'SessionTimeoutCount';
	OPCUA_BROWSENAME_SESSIONSDIAGNOSTICSSUMMARY : STRING := 'SessionsDiagnosticsSummary';
	OPCUA_BROWSENAME_SESSIONSDIAGNOSTICSSUMMARYTYPE : STRING := 'SessionsDiagnosticsSummaryType';
	OPCUA_BROWSENAME_SETADMINPASSWORD : STRING := 'SetAdminPassword';
	OPCUA_BROWSENAME_SETMONITORINGMODECOUNT : STRING := 'SetMonitoringModeCount';
	OPCUA_BROWSENAME_SETPOSITION : STRING := 'SetPosition';
	OPCUA_BROWSENAME_SETPUBLISHINGMODECOUNT : STRING := 'SetPublishingModeCount';
	OPCUA_BROWSENAME_SETREGISTRARENDPOINTS : STRING := 'SetRegistrarEndpoints';
	OPCUA_BROWSENAME_SETSECURITYKEYS : STRING := 'SetSecurityKeys';
	OPCUA_BROWSENAME_SETSUBSCRIPTIONDURABLE : STRING := 'SetSubscriptionDurable';
	OPCUA_BROWSENAME_SETTRIGGERINGCOUNT : STRING := 'SetTriggeringCount';
	OPCUA_BROWSENAME_SETPOINTNODE : STRING := 'SetpointNode';
	OPCUA_BROWSENAME_SEVERITY : STRING := 'Severity';
	OPCUA_BROWSENAME_SEVERITYHIGH : STRING := 'SeverityHigh';
	OPCUA_BROWSENAME_SEVERITYHIGHHIGH : STRING := 'SeverityHighHigh';
	OPCUA_BROWSENAME_SEVERITYLOW : STRING := 'SeverityLow';
	OPCUA_BROWSENAME_SEVERITYLOWLOW : STRING := 'SeverityLowLow';
	OPCUA_BROWSENAME_SHELVEDSTATEMACHINETYPE : STRING := 'ShelvedStateMachineType';
	OPCUA_BROWSENAME_SHELVINGSTATE : STRING := 'ShelvingState';
	OPCUA_BROWSENAME_SHELVINGTIME : STRING := 'ShelvingTime';
	OPCUA_BROWSENAME_SHUTDOWNREASON : STRING := 'ShutdownReason';
	OPCUA_BROWSENAME_SIGNEDSOFTWARECERTIFICATE : STRING := 'SignedSoftwareCertificate';
	OPCUA_BROWSENAME_SILENCE : STRING := 'Silence';
	OPCUA_BROWSENAME_SILENCESTATE : STRING := 'SilenceState';
	OPCUA_BROWSENAME_SIMPLEATTRIBUTEOPERAND : STRING := 'SimpleAttributeOperand';
	OPCUA_BROWSENAME_SIMPLETYPEDESCRIPTION : STRING := 'SimpleTypeDescription';
	OPCUA_BROWSENAME_SIZE : STRING := 'Size';
	OPCUA_BROWSENAME_SOFTWARECERTIFICATES : STRING := 'SoftwareCertificates';
	OPCUA_BROWSENAME_SOFTWAREVERSION : STRING := 'SoftwareVersion';
	OPCUA_BROWSENAME_SOURCEADDRESS : STRING := 'SourceAddress';
	OPCUA_BROWSENAME_SOURCENAME : STRING := 'SourceName';
	OPCUA_BROWSENAME_SOURCENODE : STRING := 'SourceNode';
	OPCUA_BROWSENAME_SOURCETIMESTAMP : STRING := 'SourceTimestamp';
	OPCUA_BROWSENAME_SPEED : STRING := 'Speed';
	OPCUA_BROWSENAME_SRCLASSID : STRING := 'SrClassId';
	OPCUA_BROWSENAME_STANDALONESUBSCRIBEDDATASETDATATYPE : STRING := 'StandaloneSubscribedDataSetDataType';
	OPCUA_BROWSENAME_PLACEHOLDER_STANDALONESUBSCRIBEDDATASETNAME : STRING := '<StandaloneSubscribedDataSetName>';
	OPCUA_BROWSENAME_STANDALONESUBSCRIBEDDATASETREFDATATYPE : STRING := 'StandaloneSubscribedDataSetRefDataType';
	OPCUA_BROWSENAME_STANDALONESUBSCRIBEDDATASETTYPE : STRING := 'StandaloneSubscribedDataSetType';
	OPCUA_BROWSENAME_STANDARDDEVIATIONPOPULATION : STRING := 'StandardDeviationPopulation';
	OPCUA_BROWSENAME_STANDARDDEVIATIONSAMPLE : STRING := 'StandardDeviationSample';
	OPCUA_BROWSENAME_START : STRING := 'Start';
	OPCUA_BROWSENAME_STARTBOUND : STRING := 'StartBound';
	OPCUA_BROWSENAME_STARTOFARCHIVE : STRING := 'StartOfArchive';
	OPCUA_BROWSENAME_STARTOFONLINEARCHIVE : STRING := 'StartOfOnlineArchive';
	OPCUA_BROWSENAME_STARTTIME : STRING := 'StartTime';
	OPCUA_BROWSENAME_STATE : STRING := 'State';
	OPCUA_BROWSENAME_STATEDISABLEDBYMETHOD : STRING := 'StateDisabledByMethod';
	OPCUA_BROWSENAME_STATEERROR : STRING := 'StateError';
	OPCUA_BROWSENAME_STATEMACHINETYPE : STRING := 'StateMachineType';
	OPCUA_BROWSENAME_STATENUMBER : STRING := 'StateNumber';
	OPCUA_BROWSENAME_STATEOPERATIONALBYMETHOD : STRING := 'StateOperationalByMethod';
	OPCUA_BROWSENAME_STATEOPERATIONALBYPARENT : STRING := 'StateOperationalByParent';
	OPCUA_BROWSENAME_STATEOPERATIONALFROMERROR : STRING := 'StateOperationalFromError';
	OPCUA_BROWSENAME_STATEPAUSEDBYPARENT : STRING := 'StatePausedByParent';
	OPCUA_BROWSENAME_STATETYPE : STRING := 'StateType';
	OPCUA_BROWSENAME_STATEVARIABLETYPE : STRING := 'StateVariableType';
	OPCUA_BROWSENAME_STATICNODEIDTYPES : STRING := 'StaticNodeIdTypes';
	OPCUA_BROWSENAME_STATICNUMERICNODEIDRANGE : STRING := 'StaticNumericNodeIdRange';
	OPCUA_BROWSENAME_STATICSTRINGNODEIDPATTERN : STRING := 'StaticStringNodeIdPattern';
	OPCUA_BROWSENAME_STATISTICALCONDITIONCLASSTYPE : STRING := 'StatisticalConditionClassType';
	OPCUA_BROWSENAME_STATUS : STRING := 'Status';
	OPCUA_BROWSENAME_STATUSCODE : STRING := 'StatusCode';
	OPCUA_BROWSENAME_STATUSCODEID : STRING := 'StatusCodeId';
	OPCUA_BROWSENAME_STATUSRESULT : STRING := 'StatusResult';
	OPCUA_BROWSENAME_STEPPED : STRING := 'Stepped';
	OPCUA_BROWSENAME_STREAMID : STRING := 'StreamId';
	OPCUA_BROWSENAME_STREAMNAME : STRING := 'StreamName';
	OPCUA_BROWSENAME_STREAMS : STRING := 'Streams';
	OPCUA_BROWSENAME_STRING : STRING := 'String';
	OPCUA_BROWSENAME_STRUCTURE : STRING := 'Structure';
	OPCUA_BROWSENAME_STRUCTUREDEFINITION : STRING := 'StructureDefinition';
	OPCUA_BROWSENAME_STRUCTUREDESCRIPTION : STRING := 'StructureDescription';
	OPCUA_BROWSENAME_STRUCTUREFIELD : STRING := 'StructureField';
	OPCUA_BROWSENAME_STRUCTURETYPE : STRING := 'StructureType';
	OPCUA_BROWSENAME_PLACEHOLDER_SUBALIASNAMECATEGORIES : STRING := '<SubAliasNameCategories>';
	OPCUA_BROWSENAME_SUBERROR : STRING := 'SubError';
	OPCUA_BROWSENAME_SUBSCRIBEDDATASET : STRING := 'SubscribedDataSet';
	OPCUA_BROWSENAME_SUBSCRIBEDDATASETDATATYPE : STRING := 'SubscribedDataSetDataType';
	OPCUA_BROWSENAME_PLACEHOLDER_SUBSCRIBEDDATASETFOLDERNAME : STRING := '<SubscribedDataSetFolderName>';
	OPCUA_BROWSENAME_SUBSCRIBEDDATASETFOLDERTYPE : STRING := 'SubscribedDataSetFolderType';
	OPCUA_BROWSENAME_SUBSCRIBEDDATASETMIRRORDATATYPE : STRING := 'SubscribedDataSetMirrorDataType';
	OPCUA_BROWSENAME_SUBSCRIBEDDATASETMIRRORTYPE : STRING := 'SubscribedDataSetMirrorType';
	OPCUA_BROWSENAME_SUBSCRIBEDDATASETTYPE : STRING := 'SubscribedDataSetType';
	OPCUA_BROWSENAME_SUBSCRIBEDDATASETS : STRING := 'SubscribedDataSets';
	OPCUA_BROWSENAME_SUBSCRIPTIONDIAGNOSTICS : STRING := 'SubscriptionDiagnostics';
	OPCUA_BROWSENAME_SUBSCRIPTIONDIAGNOSTICSARRAY : STRING := 'SubscriptionDiagnosticsArray';
	OPCUA_BROWSENAME_SUBSCRIPTIONDIAGNOSTICSARRAYTYPE : STRING := 'SubscriptionDiagnosticsArrayType';
	OPCUA_BROWSENAME_SUBSCRIPTIONDIAGNOSTICSDATATYPE : STRING := 'SubscriptionDiagnosticsDataType';
	OPCUA_BROWSENAME_SUBSCRIPTIONDIAGNOSTICSTYPE : STRING := 'SubscriptionDiagnosticsType';
	OPCUA_BROWSENAME_SUBSCRIPTIONID : STRING := 'SubscriptionId';
	OPCUA_BROWSENAME_SUPERVISOR : STRING := 'Supervisor';
	OPCUA_BROWSENAME_SUPPORTSECURITYKEYPULL : STRING := 'SupportSecurityKeyPull';
	OPCUA_BROWSENAME_SUPPORTSECURITYKEYPUSH : STRING := 'SupportSecurityKeyPush';
	OPCUA_BROWSENAME_SUPPORTEDPRIVATEKEYFORMATS : STRING := 'SupportedPrivateKeyFormats';
	OPCUA_BROWSENAME_SUPPORTEDSECURITYPOLICYURIS : STRING := 'SupportedSecurityPolicyUris';
	OPCUA_BROWSENAME_SUPPORTEDTRANSPORTPROFILES : STRING := 'SupportedTransportProfiles';
	OPCUA_BROWSENAME_SUPPORTSFILTEREDRETAIN : STRING := 'SupportsFilteredRetain';
	OPCUA_BROWSENAME_SUPPRESS : STRING := 'Suppress';
	OPCUA_BROWSENAME_SUPPRESS2 : STRING := 'Suppress2';
	OPCUA_BROWSENAME_SUPPRESSEDORSHELVED : STRING := 'SuppressedOrShelved';
	OPCUA_BROWSENAME_SUPPRESSEDSTATE : STRING := 'SuppressedState';
	OPCUA_BROWSENAME_SUSPEND : STRING := 'Suspend';
	OPCUA_BROWSENAME_SUSPENDED : STRING := 'Suspended';
	OPCUA_BROWSENAME_SUSPENDEDTOHALTED : STRING := 'SuspendedToHalted';
	OPCUA_BROWSENAME_SUSPENDEDTOREADY : STRING := 'SuspendedToReady';
	OPCUA_BROWSENAME_SUSPENDEDTORUNNING : STRING := 'SuspendedToRunning';
	OPCUA_BROWSENAME_SYSTEMCONDITIONCLASSTYPE : STRING := 'SystemConditionClassType';
	OPCUA_BROWSENAME_SYSTEMDIAGNOSTICALARMTYPE : STRING := 'SystemDiagnosticAlarmType';
	OPCUA_BROWSENAME_SYSTEMEVENTTYPE : STRING := 'SystemEventType';
	OPCUA_BROWSENAME_SYSTEMOFFNORMALALARMTYPE : STRING := 'SystemOffNormalAlarmType';
	OPCUA_BROWSENAME_SYSTEMSTATE : STRING := 'SystemState';
	OPCUA_BROWSENAME_SYSTEMSTATUSCHANGEEVENTTYPE : STRING := 'SystemStatusChangeEventType';
	OPCUA_BROWSENAME_TAGVARIABLES : STRING := 'TagVariables';
	OPCUA_BROWSENAME_TALKERSTATUS : STRING := 'TalkerStatus';
	OPCUA_BROWSENAME_TALKERSTREAMS : STRING := 'TalkerStreams';
	OPCUA_BROWSENAME_TARGETVALUENODE : STRING := 'TargetValueNode';
	OPCUA_BROWSENAME_TARGETVARIABLES : STRING := 'TargetVariables';
	OPCUA_BROWSENAME_TARGETVARIABLESDATATYPE : STRING := 'TargetVariablesDataType';
	OPCUA_BROWSENAME_TARGETVARIABLESTYPE : STRING := 'TargetVariablesType';
	OPCUA_BROWSENAME_TEMPORARYFILETRANSFERTYPE : STRING := 'TemporaryFileTransferType';
	OPCUA_BROWSENAME_TESTINGCONDITIONCLASSTYPE : STRING := 'TestingConditionClassType';
	OPCUA_BROWSENAME_TIME : STRING := 'Time';
	OPCUA_BROWSENAME_TIMEAVERAGE : STRING := 'TimeAverage';
	OPCUA_BROWSENAME_TIMEAVERAGE2 : STRING := 'TimeAverage2';
	OPCUA_BROWSENAME_TIMEAWAREOFFSET : STRING := 'TimeAwareOffset';
	OPCUA_BROWSENAME_TIMEFIRSTCHANGE : STRING := 'TimeFirstChange';
	OPCUA_BROWSENAME_TIMESTRING : STRING := 'TimeString';
	OPCUA_BROWSENAME_TIMETONEXTTOKENID : STRING := 'TimeToNextTokenID';
	OPCUA_BROWSENAME_TIMEZONEDATATYPE : STRING := 'TimeZoneDataType';
	OPCUA_BROWSENAME_TIMEDSHELVE : STRING := 'TimedShelve';
	OPCUA_BROWSENAME_TIMEDSHELVE2 : STRING := 'TimedShelve2';
	OPCUA_BROWSENAME_TIMEDSHELVED : STRING := 'TimedShelved';
	OPCUA_BROWSENAME_TIMEDSHELVEDTOONESHOTSHELVED : STRING := 'TimedShelvedToOneShotShelved';
	OPCUA_BROWSENAME_TIMEDSHELVEDTOUNSHELVED : STRING := 'TimedShelvedToUnshelved';
	OPCUA_BROWSENAME_TITLE : STRING := 'Title';
	OPCUA_BROWSENAME_TOSTATE : STRING := 'ToState';
	OPCUA_BROWSENAME_TOLERANCE : STRING := 'Tolerance';
	OPCUA_BROWSENAME_TOPIC : STRING := 'Topic';
	OPCUA_BROWSENAME_TOPICS : STRING := 'Topics';
	OPCUA_BROWSENAME_TOTAL : STRING := 'Total';
	OPCUA_BROWSENAME_TOTAL2 : STRING := 'Total2';
	OPCUA_BROWSENAME_TOTALERROR : STRING := 'TotalError';
	OPCUA_BROWSENAME_TOTALINFORMATION : STRING := 'TotalInformation';
	OPCUA_BROWSENAME_TOTALREQUESTCOUNT : STRING := 'TotalRequestCount';
	OPCUA_BROWSENAME_TRAININGCONDITIONCLASSTYPE : STRING := 'TrainingConditionClassType';
	OPCUA_BROWSENAME_TRANSACTIONDIAGNOSTICS : STRING := 'TransactionDiagnostics';
	OPCUA_BROWSENAME_TRANSACTIONDIAGNOSTICSTYPE : STRING := 'TransactionDiagnosticsType';
	OPCUA_BROWSENAME_TRANSACTIONERRORTYPE : STRING := 'TransactionErrorType';
	OPCUA_BROWSENAME_TRANSFERREQUESTCOUNT : STRING := 'TransferRequestCount';
	OPCUA_BROWSENAME_PLACEHOLDER_TRANSFERSTATE : STRING := '<TransferState>';
	OPCUA_BROWSENAME_TRANSFERSUBSCRIPTIONSCOUNT : STRING := 'TransferSubscriptionsCount';
	OPCUA_BROWSENAME_TRANSFERREDTOALTCLIENTCOUNT : STRING := 'TransferredToAltClientCount';
	OPCUA_BROWSENAME_TRANSFERREDTOSAMECLIENTCOUNT : STRING := 'TransferredToSameClientCount';
	OPCUA_BROWSENAME_TRANSITION : STRING := 'Transition';
	OPCUA_BROWSENAME_TRANSITIONEVENTTYPE : STRING := 'TransitionEventType';
	OPCUA_BROWSENAME_TRANSITIONNUMBER : STRING := 'TransitionNumber';
	OPCUA_BROWSENAME_TRANSITIONTIME : STRING := 'TransitionTime';
	OPCUA_BROWSENAME_TRANSITIONTYPE : STRING := 'TransitionType';
	OPCUA_BROWSENAME_TRANSITIONVARIABLETYPE : STRING := 'TransitionVariableType';
	OPCUA_BROWSENAME_TRANSLATEBROWSEPATHSTONODEIDSCOUNT : STRING := 'TranslateBrowsePathsToNodeIdsCount';
	OPCUA_BROWSENAME_TRANSMITQOSDATATYPE : STRING := 'TransmitQosDataType';
	OPCUA_BROWSENAME_TRANSMITQOSPRIORITYDATATYPE : STRING := 'TransmitQosPriorityDataType';
	OPCUA_BROWSENAME_TRANSPARENTREDUNDANCYTYPE : STRING := 'TransparentRedundancyType';
	OPCUA_BROWSENAME_TRANSPORTPROFILEURI : STRING := 'TransportProfileUri';
	OPCUA_BROWSENAME_TRANSPORTPROTOCOL : STRING := 'TransportProtocol';
	OPCUA_BROWSENAME_TRANSPORTSETTINGS : STRING := 'TransportSettings';
	OPCUA_BROWSENAME_TREATUNCERTAINASBAD : STRING := 'TreatUncertainAsBad';
	OPCUA_BROWSENAME_TRIGGERKEYUPDATE : STRING := 'TriggerKeyUpdate';
	OPCUA_BROWSENAME_TRIMMEDSTRING : STRING := 'TrimmedString';
	OPCUA_BROWSENAME_TRIPALARMTYPE : STRING := 'TripAlarmType';
	OPCUA_BROWSENAME_TRUESTATE : STRING := 'TrueState';
	OPCUA_BROWSENAME_TRUSTLIST : STRING := 'TrustList';
	OPCUA_BROWSENAME_TRUSTLISTDATATYPE : STRING := 'TrustListDataType';
	OPCUA_BROWSENAME_TRUSTLISTID : STRING := 'TrustListId';
	OPCUA_BROWSENAME_TRUSTLISTMASKS : STRING := 'TrustListMasks';
	OPCUA_BROWSENAME_TRUSTLISTOUTOFDATE : STRING := 'TrustListOutOfDate';
	OPCUA_BROWSENAME_TRUSTLISTOUTOFDATEALARMTYPE : STRING := 'TrustListOutOfDateAlarmType';
	OPCUA_BROWSENAME_TRUSTLISTTYPE : STRING := 'TrustListType';
	OPCUA_BROWSENAME_TRUSTLISTUPDATEREQUESTEDAUDITEVENTTYPE : STRING := 'TrustListUpdateRequestedAuditEventType';
	OPCUA_BROWSENAME_TRUSTLISTUPDATEDAUDITEVENTTYPE : STRING := 'TrustListUpdatedAuditEventType';
	OPCUA_BROWSENAME_TRUSTLISTVALIDATIONOPTIONS : STRING := 'TrustListValidationOptions';
	OPCUA_BROWSENAME_TSNFAILURECODE : STRING := 'TsnFailureCode';
	OPCUA_BROWSENAME_TSNLISTENERSTATUS : STRING := 'TsnListenerStatus';
	OPCUA_BROWSENAME_TSNSTREAMSTATE : STRING := 'TsnStreamState';
	OPCUA_BROWSENAME_TSNTALKERSTATUS : STRING := 'TsnTalkerStatus';
	OPCUA_BROWSENAME_TWOSTATEDISCRETETYPE : STRING := 'TwoStateDiscreteType';
	OPCUA_BROWSENAME_TWOSTATEVARIABLETYPE : STRING := 'TwoStateVariableType';
	OPCUA_BROWSENAME_TYPES : STRING := 'Types';
	OPCUA_BROWSENAME_UABINARYFILEDATATYPE : STRING := 'UABinaryFileDataType';
	OPCUA_BROWSENAME_UINT16 : STRING := 'UInt16';
	OPCUA_BROWSENAME_UINT32 : STRING := 'UInt32';
	OPCUA_BROWSENAME_UINT64 : STRING := 'UInt64';
	OPCUA_BROWSENAME_UINTEGER : STRING := 'UInteger';
	OPCUA_BROWSENAME_UADPDATASETMESSAGECONTENTMASK : STRING := 'UadpDataSetMessageContentMask';
	OPCUA_BROWSENAME_UADPDATASETREADERMESSAGEDATATYPE : STRING := 'UadpDataSetReaderMessageDataType';
	OPCUA_BROWSENAME_UADPDATASETREADERMESSAGETYPE : STRING := 'UadpDataSetReaderMessageType';
	OPCUA_BROWSENAME_UADPDATASETWRITERMESSAGEDATATYPE : STRING := 'UadpDataSetWriterMessageDataType';
	OPCUA_BROWSENAME_UADPDATASETWRITERMESSAGETYPE : STRING := 'UadpDataSetWriterMessageType';
	OPCUA_BROWSENAME_UADPNETWORKMESSAGECONTENTMASK : STRING := 'UadpNetworkMessageContentMask';
	OPCUA_BROWSENAME_UADPWRITERGROUPMESSAGEDATATYPE : STRING := 'UadpWriterGroupMessageDataType';
	OPCUA_BROWSENAME_UADPWRITERGROUPMESSAGETYPE : STRING := 'UadpWriterGroupMessageType';
	OPCUA_BROWSENAME_UNACKNOWLEDGEDCOUNT : STRING := 'UnacknowledgedCount';
	OPCUA_BROWSENAME_UNACKNOWLEDGEDMESSAGECOUNT : STRING := 'UnacknowledgedMessageCount';
	OPCUA_BROWSENAME_UNAUTHORIZEDREQUESTCOUNT : STRING := 'UnauthorizedRequestCount';
	OPCUA_BROWSENAME_UNCONFIRMEDCOUNT : STRING := 'UnconfirmedCount';
	OPCUA_BROWSENAME_UNION : STRING := 'Union';
	OPCUA_BROWSENAME_UNREGISTERNODESCOUNT : STRING := 'UnregisterNodesCount';
	OPCUA_BROWSENAME_UNSHELVE : STRING := 'Unshelve';
	OPCUA_BROWSENAME_UNSHELVE2 : STRING := 'Unshelve2';
	OPCUA_BROWSENAME_UNSHELVETIME : STRING := 'UnshelveTime';
	OPCUA_BROWSENAME_UNSHELVED : STRING := 'Unshelved';
	OPCUA_BROWSENAME_UNSHELVEDTOONESHOTSHELVED : STRING := 'UnshelvedToOneShotShelved';
	OPCUA_BROWSENAME_UNSHELVEDTOTIMEDSHELVED : STRING := 'UnshelvedToTimedShelved';
	OPCUA_BROWSENAME_UNSIGNEDRATIONALNUMBER : STRING := 'UnsignedRationalNumber';
	OPCUA_BROWSENAME_UNSUPPRESS : STRING := 'Unsuppress';
	OPCUA_BROWSENAME_UNSUPPRESS2 : STRING := 'Unsuppress2';
	OPCUA_BROWSENAME_UPDATECERTIFICATE : STRING := 'UpdateCertificate';
	OPCUA_BROWSENAME_UPDATECREDENTIAL : STRING := 'UpdateCredential';
	OPCUA_BROWSENAME_UPDATEDATACAPABILITY : STRING := 'UpdateDataCapability';
	OPCUA_BROWSENAME_UPDATEEVENTCAPABILITY : STRING := 'UpdateEventCapability';
	OPCUA_BROWSENAME_UPDATEFREQUENCY : STRING := 'UpdateFrequency';
	OPCUA_BROWSENAME_UPDATEDNODE : STRING := 'UpdatedNode';
	OPCUA_BROWSENAME_URIDICTIONARYENTRYTYPE : STRING := 'UriDictionaryEntryType';
	OPCUA_BROWSENAME_URISTRING : STRING := 'UriString';
	OPCUA_BROWSENAME_URISVERSION : STRING := 'UrisVersion';
	OPCUA_BROWSENAME_URL : STRING := 'Url';
	OPCUA_BROWSENAME_USESLOPEDEXTRAPOLATION : STRING := 'UseSlopedExtrapolation';
	OPCUA_BROWSENAME_USERCONFIGURATIONMASK : STRING := 'UserConfigurationMask';
	OPCUA_BROWSENAME_USERCREDENTIALCERTIFICATETYPE : STRING := 'UserCredentialCertificateType';
	OPCUA_BROWSENAME_USERIDENTITYTOKEN : STRING := 'UserIdentityToken';
	OPCUA_BROWSENAME_USERMANAGEMENT : STRING := 'UserManagement';
	OPCUA_BROWSENAME_USERMANAGEMENTDATATYPE : STRING := 'UserManagementDataType';
	OPCUA_BROWSENAME_USERMANAGEMENTTYPE : STRING := 'UserManagementType';
	OPCUA_BROWSENAME_USERNAMEIDENTITYTOKEN : STRING := 'UserNameIdentityToken';
	OPCUA_BROWSENAME_USERTOKENPOLICY : STRING := 'UserTokenPolicy';
	OPCUA_BROWSENAME_USERTOKENTYPE : STRING := 'UserTokenType';
	OPCUA_BROWSENAME_USERWRITABLE : STRING := 'UserWritable';
	OPCUA_BROWSENAME_USERS : STRING := 'Users';
	OPCUA_BROWSENAME_USESPRIORITYMAPPINGTABLE : STRING := 'UsesPriorityMappingTable';
	OPCUA_BROWSENAME_UTCTIME : STRING := 'UtcTime';
	OPCUA_BROWSENAME_UTILIZES : STRING := 'Utilizes';
	OPCUA_BROWSENAME_VALUEASDICTIONARYENTRIES : STRING := 'ValueAsDictionaryEntries';
	OPCUA_BROWSENAME_VALUEASTEXT : STRING := 'ValueAsText';
	OPCUA_BROWSENAME_VALUEPRECISION : STRING := 'ValuePrecision';
	OPCUA_BROWSENAME_VARIABLETYPES : STRING := 'VariableTypes';
	OPCUA_BROWSENAME_VARIANCEPOPULATION : STRING := 'VariancePopulation';
	OPCUA_BROWSENAME_VARIANCESAMPLE : STRING := 'VarianceSample';
	OPCUA_BROWSENAME_VECTOR : STRING := 'Vector';
	OPCUA_BROWSENAME_VECTORTYPE : STRING := 'VectorType';
	OPCUA_BROWSENAME_VECTORUNIT : STRING := 'VectorUnit';
	OPCUA_BROWSENAME_PLACEHOLDER_VENDORCAPABILITY : STRING := '<VendorCapability>';
	OPCUA_BROWSENAME_VENDORSERVERINFO : STRING := 'VendorServerInfo';
	OPCUA_BROWSENAME_VENDORSERVERINFOTYPE : STRING := 'VendorServerInfoType';
	OPCUA_BROWSENAME_VERSIONID : STRING := 'VersionId';
	OPCUA_BROWSENAME_VERSIONTIME : STRING := 'VersionTime';
	OPCUA_BROWSENAME_VID : STRING := 'Vid';
	OPCUA_BROWSENAME_VIEWVERSION : STRING := 'ViewVersion';
	OPCUA_BROWSENAME_VIEWS : STRING := 'Views';
	OPCUA_BROWSENAME_VLANID : STRING := 'VlanId';
	OPCUA_BROWSENAME_VLANTAGCAPABLE : STRING := 'VlanTagCapable';
	OPCUA_BROWSENAME_WORSTQUALITY : STRING := 'WorstQuality';
	OPCUA_BROWSENAME_WORSTQUALITY2 : STRING := 'WorstQuality2';
	OPCUA_BROWSENAME_WRITABLE : STRING := 'Writable';
	OPCUA_BROWSENAME_WRITE : STRING := 'Write';
	OPCUA_BROWSENAME_WRITECOUNT : STRING := 'WriteCount';
	OPCUA_BROWSENAME_WRITERGROUPDATATYPE : STRING := 'WriterGroupDataType';
	OPCUA_BROWSENAME_WRITERGROUPID : STRING := 'WriterGroupId';
	OPCUA_BROWSENAME_WRITERGROUPMESSAGEDATATYPE : STRING := 'WriterGroupMessageDataType';
	OPCUA_BROWSENAME_WRITERGROUPMESSAGETYPE : STRING := 'WriterGroupMessageType';
	OPCUA_BROWSENAME_PLACEHOLDER_WRITERGROUPNAME : STRING := '<WriterGroupName>';
	OPCUA_BROWSENAME_WRITERGROUPTRANSPORTDATATYPE : STRING := 'WriterGroupTransportDataType';
	OPCUA_BROWSENAME_WRITERGROUPTRANSPORTTYPE : STRING := 'WriterGroupTransportType';
	OPCUA_BROWSENAME_WRITERGROUPTYPE : STRING := 'WriterGroupType';
	OPCUA_BROWSENAME_X : STRING := 'X';
	OPCUA_BROWSENAME_X509IDENTITYTOKEN : STRING := 'X509IdentityToken';
	OPCUA_BROWSENAME_XAXISDEFINITION : STRING := 'XAxisDefinition';
	OPCUA_BROWSENAME_XMLSCHEMA : STRING := 'XML Schema';
	OPCUA_BROWSENAME_XVTYPE : STRING := 'XVType';
	OPCUA_BROWSENAME_XYARRAYITEMTYPE : STRING := 'XYArrayItemType';
	OPCUA_BROWSENAME_XMLELEMENT : STRING := 'XmlElement';
	OPCUA_BROWSENAME_Y : STRING := 'Y';
	OPCUA_BROWSENAME_YARRAYITEMTYPE : STRING := 'YArrayItemType';
	OPCUA_BROWSENAME_YAXISDEFINITION : STRING := 'YAxisDefinition';
	OPCUA_BROWSENAME_Z : STRING := 'Z';
	OPCUA_BROWSENAME_ZAXISDEFINITION : STRING := 'ZAxisDefinition';
END_VAR
